C01836=1155.054,198.097,-61.668,-178.059,7.198,148.783
C01837=1155.049,198.346,-61.692,-178.056,7.200,148.783
C01838=1155.045,198.596,-61.716,-178.053,7.203,148.783
C01839=1155.041,198.844,-61.740,-178.051,7.205,148.782
C01840=1155.036,199.093,-61.764,-178.048,7.208,148.782
C01841=1155.031,199.342,-61.788,-178.045,7.210,148.782
C01842=1155.027,199.590,-61.812,-178.042,7.213,148.782
C01843=1155.022,199.839,-61.836,-178.040,7.214,148.781
C01844=1155.018,200.088,-61.860,-178.037,7.217,148.781
C01845=1155.013,200.337,-61.885,-178.034,7.219,148.781
C01846=1155.009,200.585,-61.909,-178.032,7.222,148.781
C01847=1155.004,200.834,-61.932,-178.029,7.224,148.780
C01848=1155.000,201.083,-61.956,-178.026,7.227,148.780
C01849=1154.995,201.332,-61.981,-178.023,7.228,148.780
C01850=1154.991,201.581,-62.005,-178.021,7.231,148.780
C01851=1154.986,201.829,-62.029,-178.018,7.233,148.780
C01852=1154.981,202.078,-62.053,-178.015,7.236,148.779
C01853=1154.977,202.328,-62.078,-178.012,7.238,148.779
C01854=1154.973,202.576,-62.102,-178.010,7.241,148.779
C01855=1154.968,202.825,-62.127,-178.007,7.242,148.779
C01856=1154.963,203.073,-62.151,-178.004,7.245,148.779
C01857=1154.959,203.321,-62.175,-178.001,7.248,148.778
C01858=1154.954,203.572,-62.199,-177.999,7.250,148.778
C01859=1154.950,203.820,-62.223,-177.995,7.253,148.778
C01860=1154.945,204.068,-62.247,-177.993,7.255,148.778
C01861=1154.941,204.318,-62.272,-177.990,7.257,148.777
C01862=1154.936,204.566,-62.296,-177.988,7.259,148.777
C01863=1154.931,204.815,-62.321,-177.985,7.262,148.777
C01864=1154.927,205.063,-62.345,-177.982,7.264,148.777
C01865=1154.923,205.312,-62.369,-177.979,7.267,148.776
C01866=1154.918,205.561,-62.394,-177.977,7.269,148.776
C01867=1154.913,205.810,-62.418,-177.974,7.271,148.776
C01868=1154.909,206.059,-62.443,-177.971,7.273,148.776
C01869=1154.904,206.307,-62.467,-177.968,7.276,148.776
C01870=1154.899,206.556,-62.492,-177.965,7.279,148.775
C01871=1154.895,206.805,-62.516,-177.963,7.281,148.775
C01872=1154.890,207.054,-62.541,-177.960,7.284,148.775
C01873=1154.886,207.302,-62.565,-177.957,7.285,148.775
C01874=1154.881,207.551,-62.590,-177.954,7.288,148.775
C01875=1154.877,207.800,-62.614,-177.952,7.290,148.774
C01876=1154.872,208.049,-62.639,-177.949,7.293,148.774
C01877=1154.868,208.297,-62.664,-177.946,7.295,148.774
C01878=1154.863,208.546,-62.689,-177.943,7.298,148.774
C01879=1154.859,208.795,-62.713,-177.941,7.301,148.774
C01880=1154.854,209.044,-62.738,-177.938,7.302,148.773
C01881=1154.849,209.293,-62.763,-177.935,7.305,148.773
C01882=1154.844,209.563,-62.789,-177.932,7.308,148.773
C01883=1154.840,209.834,-62.816,-177.930,7.310,148.773
C01884=1154.834,210.104,-62.843,-177.926,7.312,148.772
C01885=1154.830,210.375,-62.870,-177.923,7.315,148.772
C01886=1154.825,210.623,-62.894,-177.920,7.318,148.772
C01887=1154.821,210.873,-62.919,-177.918,7.320,148.772
C01888=1154.816,211.121,-62.945,-177.915,7.323,148.772
C01889=1154.812,211.369,-62.969,-177.912,7.326,148.771
C01890=1154.807,211.619,-62.994,-177.910,7.327,148.771
C01891=1154.803,211.866,-63.019,-177.907,7.330,148.771
C01892=1154.799,212.116,-63.044,-177.904,7.332,148.771
C01893=1154.793,212.365,-63.068,-177.901,7.335,148.771
C01894=1154.789,212.612,-63.093,-177.898,7.338,148.770
C01895=1154.785,212.862,-63.118,-177.896,7.340,148.770
C01896=1154.780,213.110,-63.143,-177.893,7.343,148.770
C01897=1154.775,213.359,-63.169,-177.890,7.344,148.770
C01898=1154.771,213.608,-63.193,-177.888,7.347,148.770
C01899=1154.767,213.857,-63.218,-177.885,7.350,148.769
C01900=1154.762,214.105,-63.243,-177.882,7.352,148.769
C01901=1154.758,214.354,-63.267,-177.879,7.355,148.769
C01902=1154.753,214.602,-63.293,-177.877,7.357,148.769
C01903=1154.749,214.852,-63.318,-177.874,7.360,148.769
C01904=1154.744,215.100,-63.343,-177.871,7.363,148.769
C01905=1154.740,215.349,-63.368,-177.868,7.364,148.768
C01906=1154.735,215.597,-63.393,-177.866,7.367,148.768
C01907=1154.731,215.847,-63.418,-177.863,7.369,148.768
C01908=1154.726,216.095,-63.443,-177.860,7.372,148.768
C01909=1154.722,216.344,-63.468,-177.857,7.375,148.768
C01910=1154.717,216.592,-63.493,-177.855,7.377,148.767
C01911=1154.713,216.841,-63.518,-177.852,7.380,148.767
C01912=1154.708,217.089,-63.544,-177.849,7.382,148.767
C01913=1154.703,217.339,-63.569,-177.846,7.384,148.767
C01914=1154.698,217.587,-63.594,-177.844,7.387,148.767
C01915=1154.695,217.835,-63.619,-177.840,7.390,148.766
C01916=1154.690,218.085,-63.644,-177.838,7.392,148.766
C01917=1154.686,218.333,-63.670,-177.835,7.395,148.766
C01918=1154.681,218.582,-63.695,-177.833,7.397,148.766
C01919=1154.676,218.831,-63.720,-177.830,7.399,148.766
C01920=1154.672,219.079,-63.746,-177.827,7.402,148.766
C01921=1154.667,219.327,-63.771,-177.824,7.404,148.765
C01922=1154.663,219.577,-63.796,-177.822,7.407,148.765
C01923=1154.659,219.825,-63.821,-177.819,7.410,148.765
C01924=1154.654,220.073,-63.847,-177.816,7.412,148.765
C01925=1154.650,220.323,-63.872,-177.813,7.415,148.765
C01926=1154.645,220.571,-63.897,-177.811,7.418,148.765
C01927=1154.641,220.820,-63.923,-177.808,7.419,148.764
C01928=1154.637,221.069,-63.949,-177.805,7.422,148.764
C01929=1154.631,221.317,-63.973,-177.802,7.425,148.764
C01930=1154.627,221.566,-63.999,-177.800,7.427,148.764
C01931=1154.623,221.815,-64.025,-177.797,7.430,148.764
C01932=1154.618,222.063,-64.050,-177.794,7.433,148.763
C01933=1154.614,222.312,-64.076,-177.792,7.435,148.763
C01934=1154.609,222.560,-64.101,-177.789,7.438,148.763
C01935=1154.605,222.809,-64.127,-177.786,7.441,148.763
C01936=1154.600,223.058,-64.152,-177.783,7.442,148.763
C01937=1154.595,223.306,-64.178,-177.780,7.445,148.763
C01938=1154.591,223.555,-64.203,-177.778,7.448,148.762
C01939=1154.587,223.804,-64.229,-177.775,7.450,148.762
C01940=1154.582,224.052,-64.255,-177.772,7.453,148.762
C01941=1154.578,224.301,-64.280,-177.769,7.456,148.762
C01942=1154.574,224.550,-64.306,-177.766,7.458,148.762
C01943=1154.570,224.798,-64.332,-177.764,7.460,148.762
C01944=1154.565,225.047,-64.357,-177.761,7.463,148.761
C01945=1154.560,225.296,-64.384,-177.758,7.466,148.761
C01946=1154.556,225.544,-64.409,-177.756,7.468,148.761
C01947=1154.551,225.793,-64.435,-177.753,7.471,148.761
C01948=1154.546,226.041,-64.460,-177.750,7.474,148.761
C01949=1154.542,226.290,-64.486,-177.748,7.476,148.761
C01950=1154.538,226.539,-64.512,-177.745,7.479,148.760
C01951=1154.533,226.787,-64.537,-177.742,7.482,148.760
C01952=1154.529,227.036,-64.563,-177.739,7.484,148.760
C01953=1154.524,227.285,-64.589,-177.737,7.486,148.760
C01954=1154.520,227.534,-64.615,-177.734,7.489,148.760
C01955=1154.515,227.782,-64.641,-177.731,7.492,148.760
C01956=1154.511,228.031,-64.666,-177.728,7.494,148.759
C01957=1154.507,228.279,-64.693,-177.725,7.497,148.759
C01958=1154.502,228.528,-64.719,-177.723,7.500,148.759
C01959=1154.497,228.776,-64.744,-177.720,7.503,148.759
C01960=1154.493,229.025,-64.770,-177.717,7.505,148.759
C01961=1154.489,229.274,-64.796,-177.714,7.507,148.759
C01962=1154.484,229.523,-64.822,-177.712,7.510,148.759
C01963=1154.480,229.771,-64.849,-177.709,7.513,148.759
C01964=1154.475,230.019,-64.874,-177.706,7.515,148.758
C01965=1154.471,230.268,-64.900,-177.703,7.518,148.758
C01966=1154.466,230.517,-64.926,-177.701,7.521,148.758
C01967=1154.462,230.765,-64.953,-177.698,7.523,148.758
C01968=1154.458,231.014,-64.978,-177.695,7.526,148.758
C01969=1154.453,231.263,-65.004,-177.692,7.529,148.758
C01970=1154.448,231.511,-65.031,-177.690,7.532,148.758
C01971=1154.444,231.759,-65.057,-177.687,7.534,148.757
C01972=1154.440,232.008,-65.082,-177.684,7.536,148.757
C01973=1154.435,232.257,-65.109,-177.681,7.539,148.757
C01974=1154.431,232.506,-65.135,-177.679,7.542,148.757
C01975=1154.427,232.754,-65.161,-177.676,7.544,148.757
C01976=1154.422,233.003,-65.188,-177.673,7.547,148.757
C01977=1154.417,233.251,-65.213,-177.670,7.550,148.756
C01978=1154.413,233.499,-65.240,-177.668,7.553,148.756
C01979=1154.408,233.748,-65.266,-177.665,7.556,148.756
C01980=1154.404,233.997,-65.292,-177.663,7.558,148.756
C01981=1154.399,234.246,-65.319,-177.659,7.560,148.756
C01982=1154.395,234.494,-65.345,-177.657,7.563,148.756
C01983=1154.391,234.743,-65.371,-177.654,7.566,148.756
C01984=1154.386,234.992,-65.398,-177.652,7.568,148.756
C01985=1154.382,235.240,-65.424,-177.648,7.571,148.755
C01986=1154.377,235.512,-65.453,-177.646,7.574,148.755
C01987=1154.372,235.783,-65.481,-177.643,7.577,148.755
C01988=1154.367,236.055,-65.511,-177.640,7.580,148.755
C01989=1154.362,236.327,-65.539,-177.636,7.583,148.755
C01990=1154.358,236.575,-65.566,-177.634,7.585,148.755
C01991=1154.353,236.824,-65.592,-177.631,7.588,148.755
C01992=1154.349,237.073,-65.619,-177.628,7.591,148.755
C01993=1154.344,237.321,-65.646,-177.626,7.594,148.754
C01994=1154.340,237.570,-65.672,-177.622,7.597,148.754
C01995=1154.336,237.818,-65.699,-177.620,7.599,148.754
C01996=1154.332,238.067,-65.725,-177.617,7.602,148.754
C01997=1154.327,238.316,-65.751,-177.615,7.605,148.754
C01998=1154.323,238.564,-65.778,-177.612,7.608,148.754
C01999=1154.318,238.812,-65.805,-177.609,7.610,148.754
C02000=1154.314,239.061,-65.831,-177.606,7.612,148.753
C02001=1154.309,239.310,-65.858,-177.604,7.615,148.753
C02002=1154.305,239.558,-65.884,-177.601,7.618,148.753
C02003=1154.300,239.807,-65.911,-177.598,7.621,148.753
C02004=1154.296,240.056,-65.938,-177.595,7.624,148.753
C02005=1154.292,240.304,-65.964,-177.593,7.626,148.753
C02006=1154.287,240.552,-65.991,-177.590,7.629,148.753
C02007=1154.282,240.801,-66.018,-177.587,7.632,148.753
C02008=1154.278,241.049,-66.044,-177.584,7.635,148.753
C02009=1154.274,241.298,-66.071,-177.582,7.637,148.753
C02010=1154.270,241.546,-66.098,-177.579,7.640,148.752
C02011=1154.265,241.795,-66.125,-177.577,7.643,148.752
C02012=1154.260,242.043,-66.152,-177.574,7.645,148.752
C02013=1154.256,242.291,-66.178,-177.571,7.648,148.752
C02014=1154.252,242.540,-66.205,-177.568,7.651,148.752
C02015=1154.247,242.789,-66.232,-177.565,7.654,148.752
C02016=1154.242,243.037,-66.259,-177.563,7.656,148.752
C02017=1154.238,243.286,-66.285,-177.560,7.659,148.752
C02018=1154.234,243.535,-66.312,-177.557,7.662,148.752
C02019=1154.229,243.783,-66.340,-177.555,7.665,148.751
C02020=1154.226,244.032,-66.366,-177.552,7.668,148.751
C02021=1154.221,244.280,-66.393,-177.548,7.670,148.751
C02022=1154.216,244.528,-66.420,-177.546,7.673,148.751
C02023=1154.212,244.777,-66.447,-177.544,7.675,148.751
C02024=1154.207,245.025,-66.474,-177.541,7.678,148.751
C02025=1154.203,245.274,-66.501,-177.538,7.681,148.751
C02026=1154.199,245.523,-66.528,-177.535,7.684,148.751
C02027=1154.194,245.771,-66.555,-177.532,7.687,148.751
C02028=1154.190,246.020,-66.582,-177.530,7.689,148.751
C02029=1154.186,246.268,-66.609,-177.527,7.692,148.750
C02030=1154.181,246.516,-66.637,-177.525,7.695,148.750
C02031=1154.177,246.764,-66.664,-177.521,7.698,148.750
C02032=1154.172,247.013,-66.691,-177.519,7.701,148.750
C02033=1154.168,247.262,-66.718,-177.516,7.704,148.750
C02034=1154.163,247.511,-66.745,-177.513,7.707,148.750
C02035=1154.159,247.759,-66.772,-177.511,7.709,148.750
C02036=1154.155,248.007,-66.799,-177.508,7.712,148.750
C02037=1154.150,248.255,-66.826,-177.505,7.715,148.750
C02038=1154.146,248.504,-66.854,-177.503,7.718,148.750
C02039=1154.142,248.753,-66.881,-177.500,7.720,148.750
C02040=1154.137,249.001,-66.908,-177.497,7.723,148.749
C02041=1154.133,249.249,-66.936,-177.494,7.726,148.749
C02042=1154.128,249.498,-66.963,-177.491,7.729,148.749
C02043=1154.124,249.747,-66.990,-177.489,7.731,148.749
C02044=1154.119,249.995,-67.017,-177.486,7.734,148.749
C02045=1154.115,250.243,-67.045,-177.483,7.737,148.749
C02046=1154.110,250.492,-67.072,-177.480,7.740,148.749
C02047=1154.106,250.741,-67.100,-177.478,7.743,148.749
C02048=1154.102,250.989,-67.127,-177.475,7.746,148.749
C02049=1154.097,251.237,-67.154,-177.472,7.749,148.749
C02050=1154.093,251.486,-67.181,-177.469,7.752,148.749
C02051=1154.089,251.734,-67.210,-177.467,7.754,148.748
C02052=1154.084,251.983,-67.237,-177.464,7.757,148.748
C02053=1154.080,252.231,-67.264,-177.462,7.760,148.748
C02054=1154.076,252.480,-67.292,-177.459,7.763,148.748
C02055=1154.071,252.728,-67.319,-177.456,7.765,148.748
C02056=1154.067,252.976,-67.347,-177.453,7.768,148.748
C02057=1154.062,253.225,-67.374,-177.451,7.771,148.748
C02058=1154.058,253.473,-67.402,-177.448,7.774,148.748
C02059=1154.054,253.722,-67.429,-177.445,7.777,148.748
C02060=1154.049,253.970,-67.457,-177.442,7.780,148.748
C02061=1154.045,254.219,-67.484,-177.440,7.782,148.748
C02062=1154.041,254.467,-67.512,-177.437,7.785,148.748
C02063=1154.036,254.715,-67.539,-177.434,7.788,148.748
C02064=1154.032,254.964,-67.568,-177.432,7.791,148.748
C02065=1154.027,255.213,-67.595,-177.429,7.794,148.747
C02066=1154.023,255.461,-67.623,-177.426,7.797,148.747
C02067=1154.019,255.709,-67.651,-177.423,7.800,148.747
C02068=1154.014,255.958,-67.678,-177.421,7.803,148.747
C02069=1154.011,256.206,-67.706,-177.418,7.806,148.747
C02070=1154.006,256.455,-67.733,-177.415,7.809,148.747
C02071=1154.001,256.703,-67.761,-177.412,7.812,148.747
C02072=1153.997,256.952,-67.790,-177.410,7.814,148.747
C02073=1153.993,257.200,-67.817,-177.407,7.817,148.747
C02074=1153.988,257.448,-67.844,-177.404,7.820,148.747
C02075=1153.984,257.696,-67.873,-177.402,7.823,148.747
C02076=1153.979,257.945,-67.901,-177.399,7.826,148.747
C02077=1153.975,258.194,-67.928,-177.396,7.829,148.747
C02078=1153.971,258.442,-67.956,-177.393,7.831,148.747
C02079=1153.967,258.690,-67.984,-177.391,7.834,148.747
C02080=1153.962,258.939,-68.012,-177.388,7.837,148.747
C02081=1153.957,259.187,-68.040,-177.385,7.840,148.746
C02082=1153.954,259.436,-68.068,-177.383,7.844,148.747
C02083=1153.949,259.683,-68.096,-177.380,7.846,148.747
C02084=1153.945,259.932,-68.124,-177.377,7.849,148.746
C02085=1153.940,260.180,-68.152,-177.374,7.852,148.746
C02086=1153.936,260.429,-68.180,-177.372,7.855,148.746
C02087=1153.931,260.678,-68.208,-177.369,7.858,148.746
C02088=1153.928,260.926,-68.236,-177.367,7.860,148.746
C02089=1153.923,261.174,-68.264,-177.364,7.863,148.746
C02090=1153.918,261.448,-68.295,-177.361,7.867,148.746
C02091=1153.913,261.721,-68.326,-177.358,7.870,148.746
C02092=1153.909,261.994,-68.356,-177.355,7.873,148.746
C02093=1153.904,262.267,-68.388,-177.352,7.877,148.746
C02094=1153.900,262.516,-68.417,-177.349,7.880,148.746
C02095=1153.895,262.764,-68.444,-177.346,7.883,148.746
C02096=1153.892,263.012,-68.472,-177.343,7.886,148.746
C02097=1153.886,263.261,-68.501,-177.341,7.888,148.746
C02098=1153.883,263.509,-68.529,-177.338,7.891,148.746
C02099=1153.878,263.757,-68.557,-177.335,7.894,148.746
C02100=1153.874,264.006,-68.586,-177.333,7.898,148.746
C02101=1153.869,264.254,-68.614,-177.331,7.900,148.746
C02102=1153.865,264.503,-68.642,-177.328,7.903,148.746
C02103=1153.860,264.751,-68.670,-177.325,7.906,148.746
C02104=1153.856,264.999,-68.699,-177.322,7.909,148.746
C02105=1153.852,265.247,-68.726,-177.319,7.912,148.745
C02106=1153.847,265.496,-68.755,-177.317,7.914,148.745
C02107=1153.844,265.745,-68.783,-177.314,7.917,148.745
C02108=1153.839,265.993,-68.812,-177.311,7.920,148.745
C02109=1153.834,266.241,-68.841,-177.309,7.924,148.745
C02110=1153.830,266.489,-68.869,-177.306,7.927,148.745
C02111=1153.826,266.738,-68.898,-177.303,7.930,148.745
C02112=1153.821,266.986,-68.925,-177.300,7.932,148.745
C02113=1153.817,267.235,-68.954,-177.298,7.935,148.745
C02114=1153.813,267.483,-68.983,-177.295,7.938,148.745
C02115=1153.808,267.731,-69.011,-177.292,7.941,148.745
C02116=1153.804,267.980,-69.039,-177.290,7.945,148.745
C02117=1153.799,268.228,-69.068,-177.287,7.948,148.745
C02118=1153.795,268.476,-69.097,-177.284,7.950,148.745
C02119=1153.791,268.725,-69.125,-177.282,7.953,148.745
C02120=1153.786,268.973,-69.154,-177.279,7.956,148.745
C02121=1153.783,269.221,-69.182,-177.276,7.959,148.745
C02122=1153.778,269.470,-69.211,-177.273,7.962,148.745
C02123=1153.773,269.718,-69.240,-177.271,7.966,148.745
C02124=1153.770,269.966,-69.269,-177.268,7.968,148.745
C02125=1153.765,270.215,-69.297,-177.265,7.971,148.745
C02126=1153.760,270.463,-69.326,-177.263,7.974,148.745
C02127=1153.757,270.711,-69.355,-177.260,7.977,148.745
C02128=1153.752,270.960,-69.383,-177.258,7.981,148.745
C02129=1153.748,271.207,-69.412,-177.255,7.983,148.745
C02130=1153.744,271.456,-69.441,-177.252,7.986,148.745
C02131=1153.739,271.705,-69.469,-177.249,7.989,148.745
C02132=1153.735,271.952,-69.498,-177.246,7.992,148.745
C02133=1153.730,272.201,-69.527,-177.244,7.995,148.745
C02134=1153.727,272.449,-69.556,-177.241,7.999,148.745
C02135=1153.722,272.698,-69.585,-177.239,8.001,148.745
C02136=1153.717,272.946,-69.614,-177.236,8.004,148.745
C02137=1153.713,273.194,-69.643,-177.233,8.007,148.745
C02138=1153.709,273.442,-69.671,-177.231,8.011,148.745
C02139=1153.705,273.691,-69.701,-177.228,8.014,148.745
C02140=1153.700,273.939,-69.729,-177.225,8.017,148.745
C02141=1153.696,274.187,-69.759,-177.222,8.019,148.745
C02142=1153.692,274.436,-69.787,-177.220,8.022,148.745
C02143=1153.688,274.684,-69.816,-177.217,8.026,148.745
C02144=1153.683,274.931,-69.845,-177.214,8.029,148.745
C02145=1153.679,275.180,-69.874,-177.211,8.032,148.745
C02146=1153.675,275.429,-69.904,-177.208,8.035,148.745
C02147=1153.670,275.677,-69.933,-177.206,8.039,148.745
C02148=1153.667,275.926,-69.961,-177.203,8.042,148.745
C02149=1153.662,276.173,-69.990,-177.201,8.045,148.745
C02150=1153.658,276.421,-70.020,-177.198,8.047,148.745
C02151=1153.653,276.670,-70.049,-177.196,8.051,148.745
C02152=1153.649,276.918,-70.078,-177.193,8.054,148.745
C02153=1153.645,277.167,-70.107,-177.190,8.057,148.745
C02154=1153.640,277.414,-70.136,-177.187,8.060,148.745
C02155=1153.636,277.663,-70.166,-177.185,8.063,148.745
C02156=1153.632,277.911,-70.194,-177.182,8.066,148.745
C02157=1153.628,278.159,-70.223,-177.179,8.069,148.745
C02158=1153.624,278.408,-70.253,-177.177,8.072,148.745
C02159=1153.620,278.656,-70.282,-177.174,8.075,148.745
C02160=1153.615,278.904,-70.312,-177.171,8.078,148.745
C02161=1153.611,279.152,-70.341,-177.169,8.081,148.745
C02162=1153.606,279.401,-70.370,-177.166,8.084,148.745
C02163=1153.602,279.649,-70.399,-177.164,8.087,148.745
C02164=1153.598,279.897,-70.429,-177.161,8.090,148.745
C02165=1153.594,280.145,-70.458,-177.158,8.094,148.745
C02166=1153.589,280.394,-70.487,-177.155,8.097,148.745
C02167=1153.585,280.642,-70.517,-177.152,8.100,148.745
C02168=1153.581,280.890,-70.546,-177.150,8.103,148.745
C02169=1153.577,281.139,-70.576,-177.147,8.106,148.745
C02170=1153.572,281.386,-70.605,-177.145,8.109,148.745
C02171=1153.568,281.634,-70.634,-177.142,8.112,148.745
C02172=1153.564,281.883,-70.664,-177.140,8.115,148.745
C02173=1153.559,282.131,-70.694,-177.137,8.118,148.745
C02174=1153.555,282.380,-70.723,-177.134,8.121,148.745
C02175=1153.550,282.628,-70.753,-177.131,8.124,148.745
C02176=1153.546,282.876,-70.782,-177.129,8.128,148.745
C02177=1153.542,283.124,-70.812,-177.126,8.130,148.745
C02178=1153.538,283.373,-70.841,-177.123,8.133,148.745
C02179=1153.534,283.620,-70.871,-177.120,8.137,148.745
C02180=1153.530,283.868,-70.901,-177.118,8.140,148.745
C02181=1153.526,284.117,-70.930,-177.115,8.143,148.745
C02182=1153.521,284.365,-70.960,-177.113,8.147,148.746
C02183=1153.517,284.614,-70.990,-177.110,8.150,148.745
C02184=1153.512,284.862,-71.019,-177.108,8.153,148.746
C02185=1153.508,285.110,-71.049,-177.105,8.156,148.746
C02186=1153.504,285.358,-71.079,-177.102,8.159,148.746
C02187=1153.499,285.606,-71.109,-177.100,8.162,148.746
C02188=1153.495,285.855,-71.138,-177.097,8.165,148.746
C02189=1153.491,286.103,-71.168,-177.094,8.169,148.746
C02190=1153.487,286.351,-71.198,-177.091,8.172,148.746
C02191=1153.483,286.599,-71.227,-177.088,8.175,148.746
C02192=1153.478,286.847,-71.257,-177.086,8.178,148.746
C02193=1153.474,287.095,-71.288,-177.083,8.181,148.746
C02194=1153.469,287.370,-71.320,-177.081,8.184,148.746
C02195=1153.465,287.645,-71.353,-177.077,8.188,148.746
C02196=1153.460,287.921,-71.386,-177.074,8.192,148.746
C02197=1153.456,288.196,-71.420,-177.072,8.195,148.746
C02198=1153.451,288.445,-71.450,-177.069,8.198,148.746
C02199=1153.447,288.692,-71.480,-177.067,8.201,148.746
C02200=1153.443,288.941,-71.509,-177.064,8.204,148.746
C02201=1153.438,289.189,-71.539,-177.061,8.208,148.746
C02202=1153.434,289.437,-71.570,-177.058,8.211,148.746
C02203=1153.430,289.685,-71.599,-177.056,8.214,148.747
C02204=1153.425,289.933,-71.630,-177.053,8.217,148.746
C02205=1153.421,290.181,-71.659,-177.050,8.220,148.746
C02206=1153.417,290.429,-71.690,-177.048,8.224,148.747
C02207=1153.412,290.677,-71.720,-177.045,8.227,148.747
C02208=1153.409,290.926,-71.750,-177.043,8.230,148.747
C02209=1153.405,291.174,-71.780,-177.040,8.234,148.747
C02210=1153.400,291.422,-71.810,-177.037,8.237,148.747
C02211=1153.396,291.670,-71.840,-177.034,8.240,148.747
C02212=1153.391,291.918,-71.871,-177.032,8.243,148.747
C02213=1153.387,292.167,-71.900,-177.029,8.246,148.747
C02214=1153.382,292.415,-71.931,-177.027,8.249,148.747
C02215=1153.379,292.663,-71.961,-177.024,8.252,148.747
C02216=1153.375,292.911,-71.991,-177.021,8.256,148.747
C02217=1153.370,293.159,-72.021,-177.019,8.259,148.747
C02218=1153.366,293.407,-72.052,-177.016,8.262,148.747
C02219=1153.362,293.655,-72.082,-177.014,8.266,148.747
C02220=1153.358,293.903,-72.112,-177.011,8.269,148.747
C02221=1153.354,294.152,-72.143,-177.008,8.272,148.748
C02222=1153.349,294.400,-72.172,-177.006,8.275,148.748
C02223=1153.345,294.648,-72.203,-177.003,8.279,148.748
C02224=1153.341,294.895,-72.233,-177.000,8.282,148.748
C02225=1153.336,295.143,-72.264,-176.998,8.285,148.748
C02226=1153.333,295.392,-72.294,-176.995,8.288,148.748
C02227=1153.328,295.640,-72.325,-176.992,8.291,148.748
C02228=1153.324,295.888,-72.355,-176.990,8.294,148.748
C02229=1153.320,296.136,-72.386,-176.987,8.297,148.748
C02230=1153.316,296.385,-72.417,-176.984,8.301,148.748
C02231=1153.311,296.633,-72.446,-176.981,8.304,148.748
C02232=1153.307,296.881,-72.477,-176.979,8.308,148.748
C02233=1153.303,297.128,-72.507,-176.977,8.311,148.749
C02234=1153.299,297.377,-72.538,-176.974,8.314,148.749
C02235=1153.294,297.625,-72.569,-176.972,8.317,148.749
C02236=1153.290,297.873,-72.599,-176.968,8.321,148.749
C02237=1153.286,298.121,-72.630,-176.966,8.324,148.749
C02238=1153.282,298.369,-72.661,-176.963,8.327,148.749
C02239=1153.278,298.617,-72.691,-176.961,8.330,148.749
C02240=1153.273,298.865,-72.722,-176.958,8.333,148.749
C02241=1153.269,299.114,-72.753,-176.955,8.337,148.749
C02242=1153.265,299.361,-72.783,-176.953,8.340,148.749
C02243=1153.261,299.609,-72.814,-176.950,8.344,148.749
C02244=1153.256,299.857,-72.845,-176.948,8.347,148.749
C02245=1153.253,300.106,-72.875,-176.945,8.350,148.749
C02246=1153.248,300.354,-72.906,-176.942,8.353,148.749
C02247=1153.244,300.601,-72.937,-176.940,8.357,148.750
C02248=1153.240,300.850,-72.968,-176.937,8.360,148.750
C02249=1153.236,301.098,-72.998,-176.934,8.363,148.750
C02250=1153.231,301.346,-73.029,-176.932,8.366,148.750
C02251=1153.227,301.594,-73.060,-176.929,8.369,148.750
C02252=1153.223,301.842,-73.091,-176.926,8.373,148.750
C02253=1153.219,302.090,-73.121,-176.924,8.376,148.750
C02254=1153.215,302.338,-73.153,-176.921,8.380,148.750
C02255=1153.210,302.586,-73.184,-176.919,8.383,148.751
C02256=1153.206,302.835,-73.215,-176.916,8.386,148.750
C02257=1153.202,303.083,-73.246,-176.913,8.390,148.751
C02258=1153.197,303.331,-73.276,-176.911,8.393,148.751
C02259=1153.194,303.579,-73.307,-176.908,8.396,148.751
C02260=1153.190,303.826,-73.338,-176.906,8.399,148.751
C02261=1153.185,304.074,-73.369,-176.903,8.402,148.751
C02262=1153.181,304.323,-73.400,-176.900,8.406,148.751
C02263=1153.177,304.570,-73.432,-176.898,8.409,148.751
C02264=1153.173,304.819,-73.463,-176.895,8.413,148.751
C02265=1153.168,305.067,-73.494,-176.893,8.416,148.752
C02266=1153.163,305.315,-73.524,-176.890,8.419,148.752
C02267=1153.160,305.563,-73.556,-176.887,8.423,148.752
C02268=1153.156,305.810,-73.586,-176.885,8.426,148.752
C02269=1153.152,306.059,-73.618,-176.882,8.429,148.752
C02270=1153.148,306.306,-73.649,-176.880,8.433,148.752
C02271=1153.144,306.555,-73.680,-176.877,8.436,148.752
C02272=1153.139,306.802,-73.712,-176.874,8.440,148.752
C02273=1153.135,307.051,-73.743,-176.872,8.443,148.752
C02274=1153.131,307.299,-73.774,-176.869,8.446,148.752
C02275=1153.126,307.546,-73.805,-176.867,8.449,148.753
C02276=1153.122,307.795,-73.836,-176.864,8.453,148.753
C02277=1153.118,308.042,-73.868,-176.861,8.456,148.753
C02278=1153.114,308.291,-73.899,-176.859,8.459,148.753
C02279=1153.110,308.538,-73.930,-176.857,8.463,148.753
C02280=1153.106,308.787,-73.961,-176.853,8.466,148.753
C02281=1153.101,309.034,-73.993,-176.851,8.470,148.753
C02282=1153.097,309.283,-74.024,-176.849,8.473,148.754
C02283=1153.093,309.530,-74.055,-176.846,8.476,148.754
C02284=1153.089,309.778,-74.087,-176.843,8.480,148.754
C02285=1153.085,310.027,-74.118,-176.841,8.483,148.754
C02286=1153.080,310.275,-74.150,-176.838,8.486,148.754
C02287=1153.076,310.523,-74.182,-176.836,8.490,148.754
C02288=1153.072,310.771,-74.213,-176.833,8.494,148.754
C02289=1153.068,311.019,-74.245,-176.830,8.497,148.755
C02290=1153.064,311.267,-74.276,-176.828,8.500,148.755
C02291=1153.060,311.515,-74.308,-176.825,8.503,148.755
C02292=1153.056,311.762,-74.339,-176.822,8.507,148.755
C02293=1153.052,312.011,-74.370,-176.820,8.510,148.755
C02294=1153.048,312.259,-74.402,-176.817,8.513,148.755
C02295=1153.043,312.506,-74.434,-176.815,8.517,148.755
C02296=1153.039,312.755,-74.466,-176.812,8.521,148.756
C02297=1153.034,313.002,-74.497,-176.809,8.524,148.755
C02298=1153.030,313.280,-74.532,-176.806,8.528,148.756
C02299=1153.026,313.558,-74.568,-176.804,8.531,148.756
C02300=1153.021,313.834,-74.603,-176.801,8.535,148.756
C02301=1153.017,314.112,-74.639,-176.798,8.539,148.756
C02302=1153.012,314.361,-74.670,-176.796,8.542,148.756
C02303=1153.008,314.608,-74.702,-176.793,8.546,148.757
C02304=1153.004,314.856,-74.734,-176.790,8.549,148.757
C02305=1153.000,315.104,-74.766,-176.788,8.553,148.757
C02306=1152.995,315.352,-74.798,-176.785,8.556,148.757
C02307=1152.991,315.600,-74.830,-176.782,8.560,148.757
C02308=1152.988,315.848,-74.861,-176.780,8.563,148.757
C02309=1152.983,316.095,-74.893,-176.777,8.566,148.757
C02310=1152.979,316.344,-74.925,-176.775,8.569,148.758
C02311=1152.975,316.592,-74.957,-176.772,8.574,148.758
C02312=1152.971,316.839,-74.989,-176.770,8.577,148.758
C02313=1152.966,317.087,-75.021,-176.767,8.580,148.758
C02314=1152.963,317.335,-75.053,-176.764,8.584,148.758
C02315=1152.958,317.583,-75.084,-176.762,8.587,148.758
C02316=1152.954,317.831,-75.117,-176.759,8.590,148.759
C02317=1152.950,318.079,-75.149,-176.757,8.593,148.759
C02318=1152.947,318.327,-75.181,-176.754,8.598,148.759
C02319=1152.942,318.575,-75.213,-176.752,8.601,148.759
C02320=1152.938,318.823,-75.244,-176.749,8.604,148.759
C02321=1152.934,319.071,-75.276,-176.746,8.608,148.759
C02322=1152.929,319.319,-75.308,-176.744,8.611,148.760
C02323=1152.925,319.567,-75.340,-176.741,8.614,148.760
C02324=1152.921,319.815,-75.373,-176.738,8.618,148.760
C02325=1152.918,320.062,-75.405,-176.736,8.622,148.760
C02326=1152.913,320.310,-75.437,-176.734,8.625,148.760
C02327=1152.909,320.558,-75.469,-176.731,8.628,148.760
C02328=1152.905,320.806,-75.501,-176.728,8.632,148.760
C02329=1152.901,321.054,-75.533,-176.726,8.635,148.761
C02330=1152.897,321.302,-75.566,-176.723,8.639,148.761
C02331=1152.892,321.550,-75.598,-176.721,8.643,148.761
C02332=1152.889,321.798,-75.630,-176.718,8.646,148.761
C02333=1152.884,322.046,-75.662,-176.716,8.649,148.761
C02334=1152.881,322.293,-75.695,-176.713,8.653,148.762
C02335=1152.876,322.542,-75.727,-176.710,8.656,148.762
C02336=1152.872,322.789,-75.759,-176.708,8.660,148.762
C02337=1152.868,323.037,-75.792,-176.705,8.664,148.762
C02338=1152.864,323.285,-75.824,-176.703,8.667,148.762
C02339=1152.860,323.533,-75.856,-176.700,8.670,148.762
C02340=1152.856,323.781,-75.889,-176.697,8.674,148.763
C02341=1152.852,324.029,-75.921,-176.695,8.678,148.763
C02342=1152.848,324.276,-75.953,-176.693,8.681,148.763
C02343=1152.843,324.524,-75.986,-176.690,8.685,148.763
C02344=1152.839,324.772,-76.018,-176.687,8.688,148.763
C02345=1152.835,325.020,-76.051,-176.685,8.691,148.763
C02346=1152.831,325.268,-76.083,-176.682,8.695,148.764
C02347=1152.828,325.516,-76.116,-176.680,8.699,148.764
C02348=1152.823,325.764,-76.148,-176.677,8.702,148.764
C02349=1152.818,326.011,-76.181,-176.674,8.706,148.764
C02350=1152.815,326.259,-76.213,-176.672,8.709,148.764
C02351=1152.811,326.507,-76.246,-176.670,8.713,148.765
C02352=1152.806,326.755,-76.279,-176.667,8.717,148.765
C02353=1152.803,327.002,-76.311,-176.665,8.720,148.765
C02354=1152.798,327.251,-76.344,-176.662,8.723,148.765
C02355=1152.794,327.499,-76.377,-176.659,8.727,148.765
C02356=1152.791,327.746,-76.409,-176.657,8.730,148.766
C02357=1152.786,327.994,-76.442,-176.654,8.734,148.766
C02358=1152.782,328.242,-76.475,-176.651,8.738,148.766
C02359=1152.778,328.490,-76.508,-176.649,8.741,148.766
C02360=1152.774,328.737,-76.540,-176.646,8.745,148.766
C02361=1152.770,328.985,-76.573,-176.644,8.748,148.767
C02362=1152.765,329.233,-76.606,-176.642,8.751,148.767
C02363=1152.761,329.481,-76.638,-176.639,8.756,148.767
C02364=1152.758,329.728,-76.671,-176.636,8.759,148.767
C02365=1152.754,329.976,-76.704,-176.634,8.762,148.767
C02366=1152.749,330.224,-76.736,-176.631,8.766,148.768
C02367=1152.745,330.472,-76.770,-176.629,8.770,148.768
C02368=1152.741,330.720,-76.803,-176.626,8.774,148.768
C02369=1152.737,330.967,-76.835,-176.624,8.777,148.768
C02370=1152.733,331.215,-76.868,-176.621,8.780,148.769
C02371=1152.729,331.463,-76.901,-176.618,8.784,148.769
C02372=1152.725,331.711,-76.934,-176.616,8.788,148.769
C02373=1152.721,331.959,-76.967,-176.614,8.791,148.769
C02374=1152.716,332.207,-77.000,-176.611,8.795,148.769
C02375=1152.712,332.454,-77.034,-176.609,8.798,148.770
C02376=1152.709,332.702,-77.066,-176.606,8.802,148.770
C02377=1152.705,332.949,-77.099,-176.603,8.806,148.770
C02378=1152.700,333.198,-77.132,-176.601,8.809,148.770
C02379=1152.696,333.445,-77.165,-176.598,8.813,148.770
C02380=1152.692,333.693,-77.198,-176.596,8.816,148.771
C02381=1152.688,333.941,-77.231,-176.593,8.820,148.771
C02382=1152.684,334.189,-77.264,-176.591,8.824,148.771
C02383=1152.680,334.437,-77.298,-176.588,8.827,148.771
C02384=1152.676,334.685,-77.331,-176.585,8.831,148.772
C02385=1152.672,334.933,-77.364,-176.583,8.834,148.772
C02386=1152.668,335.180,-77.397,-176.580,8.838,148.772
C02387=1152.664,335.428,-77.430,-176.578,8.842,148.772
C02388=1152.659,335.676,-77.464,-176.575,8.845,148.772
C02389=1152.655,335.923,-77.497,-176.573,8.849,148.773
C02390=1152.652,336.171,-77.531,-176.570,8.852,148.773
C02391=1152.647,336.418,-77.564,-176.567,8.856,148.773
C02392=1152.643,336.666,-77.597,-176.565,8.860,148.774
C02393=1152.639,336.914,-77.630,-176.563,8.864,148.774
C02394=1152.636,337.162,-77.664,-176.560,8.867,148.774
C02395=1152.631,337.410,-77.697,-176.558,8.871,148.774
C02396=1152.627,337.658,-77.730,-176.555,8.875,148.774
C02397=1152.623,337.905,-77.764,-176.553,8.878,148.775
C02398=1152.619,338.152,-77.797,-176.550,8.882,148.775
C02399=1152.615,338.400,-77.830,-176.548,8.885,148.775
C02400=1152.611,338.648,-77.863,-176.545,8.889,148.775
C02401=1152.608,338.896,-77.897,-176.542,8.893,148.775
C02402=1152.602,339.176,-77.935,-176.539,8.897,148.776
C02403=1152.598,339.457,-77.973,-176.537,8.901,148.776
C02404=1152.594,339.736,-78.010,-176.534,8.905,148.776
C02405=1152.589,340.017,-78.049,-176.531,8.909,148.777
C02406=1152.585,340.264,-78.083,-176.529,8.913,148.777
C02407=1152.581,340.512,-78.116,-176.526,8.917,148.777
C02408=1152.577,340.759,-78.149,-176.524,8.920,148.777
C02409=1152.573,341.006,-78.183,-176.521,8.924,148.778
C02410=1152.569,341.255,-78.217,-176.518,8.927,148.778
C02411=1152.564,341.503,-78.250,-176.516,8.932,148.778
C02412=1152.561,341.750,-78.284,-176.514,8.935,148.778
C02413=1152.557,341.998,-78.317,-176.511,8.939,148.779
C02414=1152.553,342.245,-78.351,-176.508,8.942,148.779
C02415=1152.548,342.494,-78.385,-176.505,8.946,148.779
C02416=1152.545,342.741,-78.419,-176.503,8.950,148.779
C02417=1152.540,342.988,-78.452,-176.501,8.953,148.780
C02418=1152.536,343.236,-78.487,-176.498,8.957,148.780
C02419=1152.532,343.484,-78.520,-176.496,8.961,148.780
C02420=1152.528,343.731,-78.554,-176.493,8.965,148.780
C02421=1152.524,343.979,-78.587,-176.491,8.968,148.781
C02422=1152.520,344.227,-78.622,-176.488,8.972,148.781
C02423=1152.516,344.475,-78.655,-176.486,8.975,148.781
C02424=1152.512,344.722,-78.689,-176.483,8.980,148.782
C02425=1152.508,344.970,-78.723,-176.481,8.983,148.782
C02426=1152.504,345.217,-78.757,-176.478,8.987,148.782
C02427=1152.500,345.465,-78.791,-176.476,8.991,148.782
C02428=1152.496,345.713,-78.825,-176.473,8.995,148.783
C02429=1152.492,345.960,-78.859,-176.471,8.998,148.783
C02430=1152.489,346.208,-78.893,-176.468,9.002,148.783
C02431=1152.484,346.456,-78.927,-176.466,9.006,148.783
C02432=1152.480,346.703,-78.960,-176.463,9.010,148.784
C02433=1152.476,346.951,-78.995,-176.460,9.013,148.784
C02434=1152.472,347.199,-79.028,-176.458,9.017,148.784
C02435=1152.468,347.446,-79.062,-176.456,9.021,148.785
C02436=1152.464,347.694,-79.097,-176.453,9.025,148.785
C02437=1152.460,347.941,-79.131,-176.450,9.028,148.785
C02438=1152.455,348.189,-79.165,-176.448,9.032,148.785
C02439=1152.452,348.437,-79.199,-176.446,9.036,148.786
C02440=1152.447,348.685,-79.233,-176.443,9.040,148.786
C02441=1152.444,348.932,-79.268,-176.440,9.043,148.786
C02442=1152.440,349.180,-79.302,-176.438,9.047,148.787
C02443=1152.436,349.427,-79.336,-176.436,9.051,148.787
C02444=1152.432,349.675,-79.371,-176.433,9.055,148.787
C02445=1152.428,349.923,-79.404,-176.430,9.058,148.787
C02446=1152.423,350.170,-79.438,-176.428,9.062,148.788
C02447=1152.420,350.418,-79.473,-176.426,9.066,148.788
C02448=1152.415,350.665,-79.507,-176.423,9.070,148.788
C02449=1152.412,350.913,-79.541,-176.420,9.073,148.788
C02450=1152.408,351.161,-79.576,-176.418,9.078,148.789
C02451=1152.404,351.408,-79.610,-176.416,9.081,148.789
C02452=1152.400,351.656,-79.645,-176.413,9.085,148.789
C02453=1152.395,351.903,-79.679,-176.410,9.088,148.790
C02454=1152.392,352.151,-79.713,-176.408,9.093,148.790
C02455=1152.387,352.399,-79.748,-176.406,9.096,148.790
C02456=1152.384,352.646,-79.782,-176.403,9.100,148.790
C02457=1152.380,352.894,-79.816,-176.401,9.104,148.791
C02458=1152.376,353.142,-79.851,-176.398,9.108,148.791
C02459=1152.372,353.389,-79.885,-176.396,9.111,148.791
C02460=1152.368,353.637,-79.921,-176.393,9.115,148.792
C02461=1152.364,353.884,-79.955,-176.390,9.119,148.792
C02462=1152.360,354.132,-79.989,-176.388,9.123,148.792
C02463=1152.356,354.379,-80.024,-176.385,9.127,148.793
C02464=1152.352,354.627,-80.058,-176.383,9.130,148.793
C02465=1152.348,354.874,-80.093,-176.380,9.134,148.793
C02466=1152.344,355.122,-80.128,-176.378,9.138,148.794
C02467=1152.340,355.369,-80.162,-176.375,9.142,148.794
C02468=1152.336,355.617,-80.197,-176.373,9.145,148.794
C02469=1152.332,355.865,-80.231,-176.371,9.150,148.795
C02470=1152.328,356.113,-80.266,-176.368,9.153,148.795
C02471=1152.324,356.359,-80.301,-176.365,9.157,148.795
C02472=1152.320,356.607,-80.336,-176.363,9.162,148.795
C02473=1152.316,356.855,-80.370,-176.361,9.165,148.796
C02474=1152.312,357.102,-80.406,-176.358,9.169,148.796
C02475=1152.309,357.350,-80.440,-176.356,9.173,148.796
C02476=1152.304,357.597,-80.474,-176.353,9.177,148.797
C02477=1152.301,357.845,-80.510,-176.351,9.180,148.797
C02478=1152.296,358.092,-80.544,-176.348,9.184,148.797
C02479=1152.293,358.340,-80.579,-176.345,9.188,148.798
C02480=1152.289,358.588,-80.614,-176.343,9.192,148.798
C02481=1152.285,358.835,-80.649,-176.340,9.196,148.798
C02482=1152.281,359.083,-80.684,-176.337,9.200,148.799
C02483=1152.277,359.331,-80.719,-176.335,9.203,148.799
C02484=1152.273,359.577,-80.754,-176.333,9.208,148.799
C02485=1152.270,359.825,-80.788,-176.330,9.211,148.799
C02486=1152.265,360.072,-80.824,-176.328,9.216,148.800
C02487=1152.261,360.320,-80.858,-176.325,9.220,148.800
C02488=1152.258,360.568,-80.894,-176.323,9.223,148.800
C02489=1152.253,360.815,-80.928,-176.320,9.227,148.801
C02490=1152.249,361.063,-80.964,-176.317,9.231,148.801
C02491=1152.245,361.311,-80.999,-176.315,9.235,148.801
C02492=1152.241,361.558,-81.034,-176.312,9.239,148.802
C02493=1152.238,361.805,-81.069,-176.310,9.243,148.802
C02494=1152.234,362.053,-81.104,-176.308,9.247,148.802
C02495=1152.230,362.300,-81.139,-176.305,9.251,148.803
C02496=1152.226,362.548,-81.174,-176.302,9.255,148.803
C02497=1152.222,362.795,-81.209,-176.300,9.258,148.803
C02498=1152.218,363.042,-81.244,-176.297,9.263,148.804
C02499=1152.214,363.290,-81.279,-176.295,9.267,148.804
C02500=1152.211,363.538,-81.315,-176.292,9.270,148.804
C02501=1152.207,363.785,-81.350,-176.289,9.274,148.805
C02502=1152.203,364.032,-81.386,-176.287,9.279,148.805
C02503=1152.199,364.280,-81.420,-176.284,9.283,148.805
C02504=1152.195,364.528,-81.456,-176.282,9.286,148.806
C02505=1152.191,364.775,-81.492,-176.279,9.291,148.806
C02506=1152.186,365.058,-81.532,-176.277,9.295,148.807
C02507=1152.182,365.341,-81.573,-176.273,9.300,148.807
C02508=1152.177,365.625,-81.613,-176.271,9.304,148.807
C02509=1152.173,365.907,-81.653,-176.267,9.309,148.808
C02510=1152.169,366.154,-81.689,-176.265,9.313,148.808
C02511=1152.165,366.403,-81.724,-176.262,9.317,148.808
C02512=1152.161,366.650,-81.760,-176.260,9.321,148.809
C02513=1152.157,366.897,-81.795,-176.258,9.325,148.809
C02514=1152.153,367.145,-81.831,-176.255,9.329,148.809
C02515=1152.150,367.392,-81.866,-176.253,9.333,148.810
C02516=1152.146,367.640,-81.902,-176.250,9.337,148.810
C02517=1152.142,367.886,-81.937,-176.248,9.341,148.811
C02518=1152.137,368.134,-81.973,-176.245,9.345,148.811
C02519=1152.134,368.382,-82.009,-176.243,9.349,148.811
C02520=1152.130,368.629,-82.044,-176.241,9.353,148.812
C02521=1152.126,368.877,-82.080,-176.238,9.357,148.812
C02522=1152.123,369.124,-82.115,-176.235,9.362,148.813
C02523=1152.118,369.371,-82.151,-176.233,9.365,148.813
C02524=1152.114,369.619,-82.187,-176.231,9.370,148.813
C02525=1152.110,369.866,-82.222,-176.228,9.374,148.814
C02526=1152.107,370.114,-82.258,-176.226,9.378,148.814
C02527=1152.102,370.361,-82.294,-176.224,9.382,148.815
C02528=1152.099,370.609,-82.330,-176.221,9.386,148.815
C02529=1152.095,370.856,-82.366,-176.219,9.390,148.816
C02530=1152.091,371.103,-82.401,-176.217,9.394,148.816
C02531=1152.086,371.351,-82.437,-176.214,9.398,148.816
C02532=1152.083,371.598,-82.472,-176.212,9.402,148.817
C02533=1152.079,371.845,-82.509,-176.209,9.406,148.817
C02534=1152.075,372.093,-82.545,-176.207,9.410,148.818
C02535=1152.071,372.340,-82.580,-176.205,9.414,148.818
C02536=1152.068,372.588,-82.616,-176.203,9.418,148.818
C02537=1152.064,372.835,-82.653,-176.200,9.423,148.819
C02538=1152.060,373.083,-82.688,-176.199,9.427,148.820
C02539=1152.056,373.330,-82.724,-176.196,9.431,148.820
C02540=1152.052,373.577,-82.761,-176.194,9.435,148.820
C02541=1152.048,373.824,-82.796,-176.192,9.439,148.821
C02542=1152.044,374.072,-82.831,-176.190,9.443,148.821
C02543=1152.040,374.319,-82.868,-176.188,9.447,148.822
C02544=1152.037,374.566,-82.904,-176.186,9.451,148.822
C02545=1152.033,374.814,-82.939,-176.184,9.455,148.823
C02546=1152.029,375.061,-82.976,-176.182,9.459,148.824
C02547=1152.025,375.308,-83.012,-176.180,9.464,148.824
C02548=1152.021,375.556,-83.049,-176.178,9.468,148.825
C02549=1152.017,375.803,-83.084,-176.176,9.471,148.825
C02550=1152.013,376.051,-83.120,-176.174,9.476,148.826
C02551=1152.010,376.298,-83.157,-176.172,9.479,148.826
C02552=1152.005,376.546,-83.193,-176.170,9.484,148.827
C02553=1152.002,376.792,-83.229,-176.168,9.488,148.827
C02554=1151.997,377.040,-83.265,-176.167,9.492,148.828
C02555=1151.994,377.287,-83.301,-176.165,9.496,148.828
C02556=1151.990,377.535,-83.338,-176.163,9.500,148.829
C02557=1151.986,377.782,-83.374,-176.161,9.504,148.830
C02558=1151.982,378.030,-83.410,-176.160,9.508,148.830
C02559=1151.979,378.277,-83.446,-176.158,9.512,148.831
C02560=1151.974,378.524,-83.483,-176.157,9.516,148.831
C02561=1151.971,378.771,-83.519,-176.155,9.520,148.832
C02562=1151.967,379.018,-83.556,-176.153,9.524,148.833
C02563=1151.963,379.266,-83.591,-176.152,9.528,148.833
C02564=1151.959,379.513,-83.628,-176.151,9.532,148.834
C02565=1151.956,379.760,-83.664,-176.149,9.536,148.835
C02566=1151.951,380.008,-83.700,-176.148,9.540,148.835
C02567=1151.948,380.255,-83.737,-176.147,9.544,148.836
C02568=1151.944,380.503,-83.774,-176.146,9.547,148.837
C02569=1151.940,380.750,-83.810,-176.144,9.551,148.837
C02570=1151.937,380.997,-83.846,-176.143,9.555,148.838
C02571=1151.932,381.244,-83.883,-176.142,9.559,148.839
C02572=1151.929,381.492,-83.919,-176.141,9.563,148.839
C02573=1151.925,381.739,-83.956,-176.140,9.566,148.840
C02574=1151.921,381.986,-83.992,-176.139,9.570,148.841
C02575=1151.917,382.233,-84.029,-176.138,9.573,148.841
C02576=1151.913,382.481,-84.065,-176.137,9.578,148.842
C02577=1151.909,382.728,-84.102,-176.136,9.581,148.843
C02578=1151.905,382.975,-84.138,-176.135,9.585,148.844
C02579=1151.901,383.222,-84.175,-176.134,9.588,148.844
C02580=1151.898,383.471,-84.211,-176.133,9.593,148.845
C02581=1151.894,383.718,-84.248,-176.133,9.596,148.846
C02582=1151.890,383.965,-84.284,-176.132,9.599,148.847
C02583=1151.886,384.212,-84.321,-176.132,9.603,148.847
C02584=1151.883,384.459,-84.357,-176.131,9.607,148.848
C02585=1151.879,384.706,-84.394,-176.130,9.610,148.849
C02586=1151.874,384.954,-84.431,-176.130,9.614,148.850
C02587=1151.871,385.201,-84.467,-176.129,9.617,148.851
C02588=1151.867,385.449,-84.504,-176.129,9.620,148.851
C02589=1151.863,385.696,-84.541,-176.129,9.623,148.852
C02590=1151.860,385.943,-84.577,-176.129,9.627,148.853
C02591=1151.856,386.190,-84.614,-176.129,9.630,148.854
C02592=1151.852,386.437,-84.651,-176.128,9.633,148.854
C02593=1151.848,386.685,-84.686,-176.129,9.636,148.855
C02594=1151.844,386.932,-84.723,-176.128,9.640,148.856
C02595=1151.840,387.179,-84.760,-176.129,9.643,148.857
C02596=1151.836,387.427,-84.797,-176.128,9.646,148.858
C02597=1151.833,387.674,-84.834,-176.129,9.649,148.859
C02598=1151.829,387.921,-84.870,-176.128,9.652,148.859
C02599=1151.825,388.168,-84.907,-176.129,9.655,148.860
C02600=1151.821,388.415,-84.944,-176.129,9.658,148.861
C02601=1151.817,388.662,-84.980,-176.129,9.660,148.862
C02602=1151.814,388.910,-85.018,-176.129,9.664,148.863
C02603=1151.810,389.157,-85.054,-176.129,9.667,148.864
C02604=1151.806,389.404,-85.091,-176.130,9.670,148.864
C02605=1151.802,389.651,-85.128,-176.130,9.672,148.865
C02606=1151.798,389.899,-85.164,-176.131,9.675,148.866
C02607=1151.794,390.146,-85.201,-176.131,9.678,148.867
C02608=1151.791,390.394,-85.237,-176.132,9.681,148.868
C02609=1151.787,390.641,-85.274,-176.132,9.683,148.869
C02610=1151.783,390.927,-85.317,-176.133,9.687,148.870
C02611=1151.778,391.213,-85.359,-176.133,9.689,148.871
C02612=1151.774,391.500,-85.402,-176.134,9.692,148.871
C02613=1151.769,391.786,-85.445,-176.135,9.695,148.873
C02614=1151.765,392.034,-85.481,-176.135,9.698,148.873
C02615=1151.761,392.281,-85.518,-176.136,9.701,148.874
C02616=1151.757,392.528,-85.555,-176.137,9.703,148.875
C02617=1151.754,392.776,-85.592,-176.137,9.706,148.876
C02618=1151.750,393.023,-85.629,-176.138,9.709,148.877
C02619=1151.746,393.270,-85.666,-176.139,9.711,148.878
C02620=1151.742,393.517,-85.702,-176.139,9.714,148.879
C02621=1151.739,393.764,-85.739,-176.140,9.716,148.879
C02622=1151.735,394.012,-85.776,-176.141,9.718,148.880
C02623=1151.731,394.259,-85.813,-176.142,9.720,148.881
C02624=1151.727,394.506,-85.850,-176.142,9.723,148.882
C02625=1151.723,394.753,-85.886,-176.143,9.725,148.883
C02626=1151.720,395.000,-85.923,-176.144,9.727,148.884
C02627=1151.715,395.247,-85.960,-176.145,9.730,148.884
C02628=1151.712,395.495,-85.997,-176.146,9.732,148.885
C02629=1151.708,395.743,-86.034,-176.147,9.734,148.886
C02630=1151.704,395.990,-86.071,-176.147,9.737,148.887
C02631=1151.700,396.237,-86.107,-176.148,9.739,148.888
C02632=1151.696,396.484,-86.144,-176.149,9.741,148.888
C02633=1151.692,396.731,-86.180,-176.151,9.743,148.889
C02634=1151.689,396.979,-86.218,-176.151,9.746,148.890
C02635=1151.685,397.226,-86.255,-176.152,9.748,148.891
C02636=1151.681,397.473,-86.291,-176.153,9.750,148.892
C02637=1151.677,397.720,-86.328,-176.154,9.752,148.893
C02638=1151.673,397.967,-86.365,-176.155,9.754,148.893
C02639=1151.670,398.215,-86.402,-176.156,9.757,148.894
C02640=1151.665,398.462,-86.439,-176.156,9.759,148.895
C02641=1151.662,398.709,-86.475,-176.157,9.761,148.896
C02642=1151.658,398.957,-86.512,-176.159,9.763,148.897
C02643=1151.654,399.204,-86.549,-176.160,9.765,148.897
C02644=1151.650,399.451,-86.585,-176.161,9.767,148.898
C02645=1151.646,399.699,-86.623,-176.161,9.769,148.899
C02646=1151.643,399.946,-86.659,-176.163,9.771,148.900
C02647=1151.639,400.193,-86.696,-176.164,9.773,148.901
C02648=1151.635,400.440,-86.733,-176.164,9.774,148.901
C02649=1151.631,400.687,-86.770,-176.166,9.776,148.902
C02650=1151.627,400.935,-86.807,-176.167,9.778,148.903
C02651=1151.624,401.182,-86.843,-176.168,9.781,148.904
C02652=1151.620,401.429,-86.881,-176.168,9.782,148.904
C02653=1151.616,401.676,-86.917,-176.170,9.784,148.905
C02654=1151.612,401.923,-86.954,-176.171,9.786,148.906
C02655=1151.608,402.171,-86.992,-176.171,9.788,148.907
C02656=1151.605,402.418,-87.028,-176.172,9.790,148.908
C02657=1151.601,402.665,-87.065,-176.174,9.792,148.908
C02658=1151.597,402.912,-87.102,-176.174,9.794,148.909
C02659=1151.593,403.159,-87.138,-176.175,9.796,148.910
C02660=1151.589,403.406,-87.175,-176.176,9.798,148.911
C02661=1151.586,403.654,-87.212,-176.177,9.800,148.911
C02662=1151.582,403.901,-87.249,-176.178,9.802,148.912
C02663=1151.578,404.148,-87.286,-176.179,9.804,148.913
C02664=1151.574,404.396,-87.322,-176.180,9.806,148.914
C02665=1151.570,404.643,-87.359,-176.181,9.808,148.914
C02666=1151.566,404.891,-87.397,-176.182,9.810,148.915
C02667=1151.563,405.138,-87.433,-176.182,9.811,148.916
C02668=1151.559,405.385,-87.470,-176.184,9.813,148.917
C02669=1151.554,405.632,-87.506,-176.184,9.815,148.917
C02670=1151.550,405.879,-87.543,-176.186,9.816,148.918
C02671=1151.547,406.127,-87.581,-176.187,9.818,148.919
C02672=1151.544,406.374,-87.617,-176.187,9.820,148.919
C02673=1151.539,406.621,-87.654,-176.188,9.822,148.920
C02674=1151.535,406.868,-87.691,-176.189,9.824,148.921
C02675=1151.531,407.116,-87.727,-176.190,9.826,148.922
C02676=1151.528,407.363,-87.765,-176.191,9.828,148.922
C02677=1151.525,407.610,-87.802,-176.192,9.829,148.923
C02678=1151.521,407.857,-87.838,-176.193,9.831,148.924
C02679=1151.517,408.104,-87.875,-176.193,9.833,148.924
C02680=1151.512,408.351,-87.912,-176.194,9.835,148.925
C02681=1151.509,408.599,-87.949,-176.195,9.837,148.926
C02682=1151.505,408.846,-87.986,-176.196,9.839,148.927
C02683=1151.501,409.093,-88.023,-176.197,9.840,148.927
C02684=1151.497,409.340,-88.059,-176.198,9.842,148.928
C02685=1151.493,409.588,-88.096,-176.198,9.844,148.929
C02686=1151.490,409.835,-88.133,-176.199,9.846,148.929
C02687=1151.486,410.083,-88.170,-176.200,9.848,148.930
C02688=1151.482,410.330,-88.207,-176.201,9.850,148.931
C02689=1151.478,410.577,-88.243,-176.201,9.852,148.931
C02690=1151.474,410.824,-88.280,-176.202,9.853,148.932
C02691=1151.470,411.071,-88.317,-176.203,9.855,148.933
C02692=1151.467,411.319,-88.354,-176.204,9.857,148.934
C02693=1151.462,411.566,-88.391,-176.205,9.859,148.934
C02694=1151.459,411.813,-88.428,-176.205,9.861,148.935
C02695=1151.455,412.060,-88.464,-176.206,9.862,148.935
C02696=1151.451,412.307,-88.502,-176.207,9.864,148.936
C02697=1151.448,412.555,-88.539,-176.207,9.867,148.937
C02698=1151.444,412.802,-88.576,-176.208,9.869,148.938
C02699=1151.440,413.049,-88.613,-176.208,9.870,148.938
C02700=1151.436,413.296,-88.649,-176.209,9.872,148.939
C02701=1151.432,413.543,-88.686,-176.210,9.874,148.940
C02702=1151.429,413.791,-88.723,-176.211,9.876,148.940
C02703=1151.425,414.038,-88.760,-176.211,9.877,148.941
C02704=1151.420,414.285,-88.797,-176.212,9.879,148.941
C02705=1151.416,414.533,-88.834,-176.213,9.881,148.942
C02706=1151.413,414.780,-88.870,-176.213,9.884,148.943
C02707=1151.409,415.027,-88.907,-176.214,9.886,148.944
C02708=1151.407,415.274,-88.945,-176.214,9.887,148.944
C02709=1151.405,415.522,-88.981,-176.215,9.889,148.945
C02710=1151.405,415.738,-89.013,-176.215,9.891,148.945
C02711=1151.404,415.955,-89.045,-176.216,9.892,148.946
C02712=1151.404,416.171,-89.077,-176.216,9.894,148.946
C02713=1151.405,416.387,-89.108,-176.217,9.895,148.947
C02714=1151.407,416.604,-89.140,-176.217,9.897,148.948
C02715=1151.408,416.820,-89.172,-176.218,9.899,148.948
C02716=1151.411,417.036,-89.203,-176.218,9.900,148.949
C02717=1151.414,417.252,-89.235,-176.218,9.902,148.949
C02718=1150.994,417.253,-89.284,-176.221,9.913,148.953
C02719=1150.990,417.036,-89.252,-176.221,9.911,148.952
C02720=1150.988,416.819,-89.220,-176.221,9.909,148.952
C02721=1150.986,416.600,-89.189,-176.220,9.908,148.951
C02722=1150.984,416.382,-89.156,-176.220,9.906,148.951
C02723=1150.984,416.165,-89.125,-176.219,9.904,148.950
C02724=1150.984,415.947,-89.092,-176.219,9.903,148.950
C02725=1150.984,415.729,-89.060,-176.218,9.901,148.949
C02726=1150.984,415.510,-89.027,-176.218,9.900,148.948
C02727=1150.986,415.263,-88.991,-176.217,9.898,148.948
C02728=1150.989,415.015,-88.955,-176.216,9.896,148.947
C02729=1150.992,414.768,-88.917,-176.215,9.894,148.946
C02730=1150.996,414.521,-88.880,-176.215,9.892,148.946
C02731=1151.000,414.274,-88.843,-176.214,9.891,148.945
C02732=1151.004,414.027,-88.807,-176.214,9.888,148.944
C02733=1151.007,413.779,-88.769,-176.213,9.886,148.944
C02734=1151.011,413.532,-88.733,-176.212,9.885,148.943
C02735=1151.016,413.285,-88.696,-176.212,9.883,148.942
C02736=1151.019,413.038,-88.659,-176.211,9.881,148.942
C02737=1151.023,412.791,-88.623,-176.210,9.879,148.941
C02738=1151.027,412.543,-88.585,-176.209,9.877,148.940
C02739=1151.031,412.295,-88.548,-176.209,9.876,148.940
C02740=1151.034,412.049,-88.511,-176.208,9.874,148.939
C02741=1151.039,411.802,-88.474,-176.207,9.872,148.938
C02742=1151.043,411.555,-88.437,-176.206,9.870,148.938
C02743=1151.045,411.307,-88.401,-176.206,9.867,148.937
C02744=1151.049,411.060,-88.364,-176.205,9.866,148.936
C02745=1151.054,410.813,-88.327,-176.205,9.864,148.936
C02746=1151.058,410.565,-88.290,-176.204,9.862,148.935
C02747=1151.062,410.318,-88.253,-176.203,9.860,148.934
C02748=1151.065,410.070,-88.216,-176.202,9.858,148.933
C02749=1151.069,409.823,-88.180,-176.202,9.857,148.933
C02750=1151.073,409.576,-88.143,-176.201,9.855,148.932
C02751=1151.077,409.329,-88.106,-176.200,9.853,148.931
C02752=1151.081,409.082,-88.069,-176.199,9.851,148.931
C02753=1151.084,408.834,-88.032,-176.198,9.849,148.930
C02754=1151.088,408.587,-87.996,-176.197,9.847,148.929
C02755=1151.092,408.341,-87.958,-176.197,9.846,148.929
C02756=1151.096,408.093,-87.921,-176.196,9.843,148.928
C02757=1151.100,407.846,-87.884,-176.195,9.842,148.927
C02758=1151.103,407.598,-87.847,-176.194,9.840,148.926
C02759=1151.107,407.351,-87.810,-176.193,9.839,148.926
C02760=1151.111,407.104,-87.774,-176.192,9.837,148.925
C02761=1151.115,406.857,-87.737,-176.191,9.835,148.924
C02762=1151.119,406.610,-87.700,-176.190,9.833,148.924
C02763=1151.122,406.362,-87.663,-176.189,9.831,148.923
C02764=1151.126,406.115,-87.626,-176.188,9.829,148.922
C02765=1151.130,405.868,-87.590,-176.188,9.828,148.921
C02766=1151.134,405.621,-87.553,-176.187,9.826,148.921
C02767=1151.138,405.373,-87.516,-176.186,9.824,148.920
C02768=1151.141,405.126,-87.479,-176.185,9.822,148.919
C02769=1151.146,404.878,-87.442,-176.184,9.820,148.918
C02770=1151.150,404.631,-87.405,-176.183,9.818,148.918
C02771=1151.153,404.384,-87.369,-176.182,9.816,148.917
C02772=1151.157,404.138,-87.331,-176.181,9.814,148.916
C02773=1151.160,403.890,-87.294,-176.180,9.812,148.915
C02774=1151.164,403.643,-87.257,-176.179,9.810,148.915
C02775=1151.168,403.395,-87.220,-176.178,9.808,148.914
C02776=1151.172,403.149,-87.184,-176.178,9.806,148.913
C02777=1151.176,402.901,-87.147,-176.176,9.805,148.912
C02778=1151.180,402.654,-87.110,-176.175,9.803,148.912
C02779=1151.184,402.406,-87.073,-176.174,9.801,148.911
C02780=1151.188,402.159,-87.036,-176.173,9.799,148.910
C02781=1151.192,401.912,-87.000,-176.172,9.797,148.909
C02782=1151.195,401.665,-86.963,-176.171,9.796,148.909
C02783=1151.199,401.418,-86.926,-176.170,9.793,148.908
C02784=1151.203,401.170,-86.889,-176.169,9.791,148.907
C02785=1151.207,400.923,-86.852,-176.168,9.790,148.906
C02786=1151.211,400.676,-86.815,-176.167,9.788,148.905
C02787=1151.214,400.429,-86.779,-176.166,9.786,148.905
C02788=1151.218,400.182,-86.742,-176.165,9.783,148.904
C02789=1151.222,399.934,-86.705,-176.164,9.782,148.903
C02790=1151.226,399.686,-86.668,-176.163,9.780,148.902
C02791=1151.230,399.439,-86.631,-176.162,9.778,148.901
C02792=1151.234,399.192,-86.595,-176.161,9.776,148.901
C02793=1151.237,398.945,-86.558,-176.161,9.773,148.900
C02794=1151.241,398.698,-86.520,-176.160,9.771,148.899
C02795=1151.245,398.451,-86.483,-176.159,9.769,148.898
C02796=1151.249,398.204,-86.447,-176.158,9.767,148.897
C02797=1151.253,397.956,-86.410,-176.156,9.765,148.897
C02798=1151.256,397.709,-86.373,-176.156,9.763,148.896
C02799=1151.260,397.462,-86.336,-176.155,9.761,148.895
C02800=1151.264,397.214,-86.299,-176.153,9.759,148.894
C02801=1151.268,396.967,-86.263,-176.153,9.756,148.893
C02802=1151.272,396.720,-86.226,-176.152,9.754,148.892
C02803=1151.275,396.473,-86.189,-176.151,9.752,148.892
C02804=1151.279,396.226,-86.153,-176.150,9.750,148.891
C02805=1151.283,395.978,-86.115,-176.150,9.747,148.890
C02806=1151.287,395.731,-86.078,-176.148,9.745,148.889
C02807=1151.291,395.484,-86.042,-176.147,9.743,148.888
C02808=1151.295,395.237,-86.005,-176.146,9.741,148.888
C02809=1151.299,394.990,-85.969,-176.146,9.738,148.887
C02810=1151.302,394.742,-85.931,-176.145,9.736,148.886
C02811=1151.306,394.494,-85.894,-176.144,9.733,148.885
C02812=1151.310,394.247,-85.858,-176.143,9.732,148.884
C02813=1151.314,394.000,-85.821,-176.142,9.729,148.883
C02814=1151.318,393.753,-85.784,-176.142,9.727,148.883
C02815=1151.322,393.506,-85.748,-176.141,9.725,148.882
C02816=1151.325,393.258,-85.710,-176.140,9.722,148.881
C02817=1151.329,393.011,-85.674,-176.139,9.720,148.880
C02818=1151.333,392.764,-85.637,-176.138,9.717,148.879
C02819=1151.337,392.517,-85.600,-176.138,9.714,148.878
C02820=1151.341,392.270,-85.564,-176.137,9.712,148.878
C02821=1151.344,392.022,-85.526,-176.137,9.709,148.877
C02822=1151.348,391.775,-85.490,-176.136,9.706,148.876
C02823=1151.353,391.488,-85.446,-176.136,9.703,148.875
C02824=1151.358,391.202,-85.404,-176.135,9.700,148.874
C02825=1151.362,390.916,-85.362,-176.134,9.697,148.873
C02826=1151.366,390.629,-85.319,-176.134,9.695,148.872
C02827=1151.370,390.383,-85.283,-176.133,9.692,148.871
C02828=1151.374,390.135,-85.246,-176.132,9.689,148.870
C02829=1151.377,389.888,-85.209,-176.132,9.686,148.869
C02830=1151.381,389.640,-85.172,-176.132,9.683,148.869
C02831=1151.385,389.393,-85.135,-176.131,9.681,148.868
C02832=1151.389,389.146,-85.099,-176.131,9.678,148.867
C02833=1151.393,388.899,-85.062,-176.131,9.675,148.866
C02834=1151.397,388.652,-85.025,-176.130,9.672,148.865
C02835=1151.400,388.404,-84.988,-176.130,9.669,148.864
C02836=1151.404,388.156,-84.952,-176.130,9.666,148.864
C02837=1151.408,387.909,-84.915,-176.130,9.663,148.863
C02838=1151.412,387.662,-84.878,-176.130,9.660,148.862
C02839=1151.416,387.415,-84.842,-176.129,9.657,148.861
C02840=1151.420,387.168,-84.805,-176.129,9.654,148.860
C02841=1151.423,386.920,-84.768,-176.129,9.651,148.859
C02842=1151.427,386.673,-84.731,-176.130,9.647,148.859
C02843=1151.431,386.426,-84.695,-176.130,9.645,148.858
C02844=1151.435,386.179,-84.658,-176.130,9.641,148.857
C02845=1151.439,385.932,-84.621,-176.130,9.638,148.856
C02846=1151.442,385.685,-84.585,-176.130,9.635,148.855
C02847=1151.447,385.437,-84.549,-176.131,9.632,148.855
C02848=1151.450,385.189,-84.512,-176.131,9.628,148.854
C02849=1151.453,384.942,-84.475,-176.131,9.625,148.853
C02850=1151.457,384.695,-84.438,-176.132,9.621,148.852
C02851=1151.462,384.448,-84.402,-176.132,9.618,148.851
C02852=1151.466,384.201,-84.365,-176.133,9.614,148.851
C02853=1151.469,383.954,-84.329,-176.134,9.610,148.850
C02854=1151.473,383.706,-84.292,-176.134,9.607,148.849
C02855=1151.478,383.459,-84.256,-176.135,9.603,148.848
C02856=1151.480,383.211,-84.219,-176.135,9.600,148.848
C02857=1151.484,382.964,-84.182,-176.137,9.596,148.847
C02858=1151.488,382.717,-84.145,-176.137,9.593,148.846
C02859=1151.492,382.469,-84.110,-176.138,9.589,148.845
C02860=1151.496,382.222,-84.073,-176.139,9.585,148.845
C02861=1151.500,381.975,-84.036,-176.140,9.581,148.844
C02862=1151.504,381.728,-84.000,-176.141,9.577,148.843
C02863=1151.508,381.480,-83.963,-176.142,9.574,148.843
C02864=1151.511,381.233,-83.927,-176.143,9.570,148.842
C02865=1151.516,380.986,-83.890,-176.144,9.566,148.841
C02866=1151.520,380.739,-83.854,-176.146,9.562,148.841
C02867=1151.523,380.491,-83.818,-176.147,9.559,148.840
C02868=1151.527,380.244,-83.781,-176.148,9.555,148.839
C02869=1151.530,379.997,-83.744,-176.149,9.551,148.839
C02870=1151.535,379.749,-83.708,-176.151,9.547,148.838
C02871=1151.538,379.502,-83.672,-176.152,9.543,148.837
C02872=1151.542,379.255,-83.635,-176.154,9.539,148.837
C02873=1151.546,379.007,-83.599,-176.155,9.535,148.836
C02874=1151.550,378.760,-83.563,-176.157,9.531,148.836
C02875=1151.554,378.512,-83.527,-176.158,9.528,148.835
C02876=1151.557,378.265,-83.490,-176.160,9.523,148.834
C02877=1151.562,378.018,-83.454,-176.162,9.519,148.834
C02878=1151.565,377.771,-83.418,-176.163,9.515,148.833
C02879=1151.569,377.524,-83.381,-176.165,9.511,148.832
C02880=1151.573,377.276,-83.346,-176.167,9.506,148.832
C02881=1151.577,377.029,-83.309,-176.169,9.503,148.831
C02882=1151.581,376.781,-83.273,-176.170,9.499,148.831
C02883=1151.585,376.534,-83.236,-176.172,9.495,148.830
C02884=1151.589,376.287,-83.201,-176.174,9.491,148.830
C02885=1151.593,376.040,-83.164,-176.176,9.487,148.829
C02886=1151.596,375.792,-83.128,-176.178,9.482,148.828
C02887=1151.600,375.545,-83.092,-176.179,9.478,148.828
C02888=1151.604,375.297,-83.056,-176.181,9.475,148.827
C02889=1151.608,375.049,-83.020,-176.184,9.471,148.827
C02890=1151.612,374.803,-82.984,-176.185,9.467,148.826
C02891=1151.615,374.555,-82.948,-176.188,9.462,148.826
C02892=1151.620,374.308,-82.911,-176.190,9.459,148.825
C02893=1151.623,374.060,-82.876,-176.192,9.454,148.825
C02894=1151.628,373.813,-82.839,-176.194,9.450,148.824
C02895=1151.631,373.566,-82.803,-176.196,9.446,148.824
C02896=1151.635,373.318,-82.768,-176.199,9.442,148.823
C02897=1151.639,373.070,-82.732,-176.200,9.438,148.823
C02898=1151.643,372.824,-82.696,-176.203,9.433,148.822
C02899=1151.647,372.577,-82.660,-176.204,9.430,148.822
C02900=1151.651,372.329,-82.624,-176.207,9.425,148.821
C02901=1151.655,372.081,-82.588,-176.209,9.421,148.821
C02902=1151.658,371.835,-82.552,-176.211,9.417,148.821
C02903=1151.662,371.587,-82.516,-176.214,9.413,148.820
C02904=1151.666,371.339,-82.480,-176.217,9.409,148.820
C02905=1151.670,371.092,-82.445,-176.219,9.405,148.819
C02906=1151.673,370.845,-82.409,-176.221,9.401,148.819
C02907=1151.678,370.597,-82.372,-176.224,9.396,148.818
C02908=1151.682,370.350,-82.337,-176.225,9.393,148.818
C02909=1151.685,370.103,-82.302,-176.228,9.388,148.818
C02910=1151.690,369.855,-82.266,-176.230,9.384,148.817
C02911=1151.694,369.607,-82.230,-176.233,9.381,148.817
C02912=1151.697,369.360,-82.194,-176.235,9.376,148.816
C02913=1151.701,369.112,-82.159,-176.238,9.372,148.816
C02914=1151.705,368.865,-82.123,-176.240,9.369,148.816
C02915=1151.710,368.618,-82.088,-176.242,9.364,148.815
C02916=1151.713,368.371,-82.051,-176.245,9.360,148.815
C02917=1151.717,368.123,-82.016,-176.248,9.356,148.814
C02918=1151.720,367.876,-81.980,-176.250,9.352,148.814
C02919=1151.724,367.628,-81.945,-176.252,9.348,148.814
C02920=1151.729,367.381,-81.910,-176.255,9.344,148.813
C02921=1151.733,367.133,-81.874,-176.257,9.340,148.813
C02922=1151.737,366.886,-81.839,-176.260,9.336,148.813
C02923=1151.740,366.638,-81.803,-176.262,9.332,148.812
C02924=1151.744,366.391,-81.767,-176.265,9.328,148.812
C02925=1151.748,366.144,-81.732,-176.267,9.324,148.811
C02926=1151.752,365.896,-81.697,-176.270,9.320,148.811
C02927=1151.756,365.613,-81.656,-176.273,9.315,148.811
C02928=1151.761,365.330,-81.615,-176.276,9.310,148.810
C02929=1151.766,365.047,-81.575,-176.279,9.306,148.810
C02930=1151.769,364.764,-81.535,-176.282,9.301,148.809
C02931=1151.773,364.516,-81.499,-176.284,9.298,148.809
C02932=1151.778,364.269,-81.465,-176.286,9.293,148.809
C02933=1151.781,364.022,-81.429,-176.289,9.289,148.808
C02934=1151.785,363.774,-81.393,-176.292,9.285,148.808
C02935=1151.789,363.527,-81.358,-176.294,9.282,148.808
C02936=1151.793,363.279,-81.323,-176.297,9.277,148.808
C02937=1151.797,363.032,-81.288,-176.300,9.273,148.807
C02938=1151.800,362.784,-81.252,-176.302,9.270,148.807
C02939=1151.805,362.537,-81.218,-176.305,9.266,148.807
C02940=1151.809,362.289,-81.182,-176.307,9.261,148.806
C02941=1151.812,362.042,-81.147,-176.310,9.258,148.806
C02942=1151.816,361.794,-81.112,-176.312,9.254,148.805
C02943=1151.821,361.547,-81.077,-176.315,9.249,148.805
C02944=1151.824,361.299,-81.041,-176.318,9.245,148.805
C02945=1151.828,361.051,-81.006,-176.320,9.242,148.804
C02946=1151.832,360.804,-80.971,-176.323,9.238,148.804
C02947=1151.836,360.556,-80.936,-176.326,9.234,148.804
C02948=1151.840,360.309,-80.901,-176.327,9.230,148.804
C02949=1151.845,360.061,-80.866,-176.330,9.226,148.803
C02950=1151.848,359.814,-80.831,-176.332,9.222,148.803
C02951=1151.852,359.567,-80.797,-176.335,9.218,148.803
C02952=1151.856,359.319,-80.761,-176.338,9.214,148.802
C02953=1151.860,359.071,-80.727,-176.340,9.211,148.802
C02954=1151.864,358.824,-80.691,-176.343,9.206,148.802
C02955=1151.868,358.576,-80.657,-176.346,9.202,148.801
C02956=1151.871,358.329,-80.622,-176.348,9.199,148.801
C02957=1151.875,358.082,-80.587,-176.351,9.195,148.801
C02958=1151.879,357.833,-80.552,-176.353,9.191,148.800
C02959=1151.884,357.587,-80.517,-176.355,9.187,148.800
C02960=1151.888,357.339,-80.482,-176.358,9.183,148.800
C02961=1151.892,357.091,-80.448,-176.360,9.179,148.799
C02962=1151.895,356.844,-80.413,-176.363,9.175,148.799
C02963=1151.899,356.596,-80.378,-176.365,9.172,148.799
C02964=1151.904,356.348,-80.344,-176.368,9.168,148.798
C02965=1151.907,356.101,-80.309,-176.370,9.164,148.798
C02966=1151.911,355.854,-80.274,-176.373,9.160,148.798
C02967=1151.915,355.606,-80.239,-176.376,9.156,148.797
C02968=1151.920,355.358,-80.205,-176.378,9.153,148.797
C02969=1151.923,355.111,-80.170,-176.381,9.148,148.797
C02970=1151.927,354.864,-80.135,-176.383,9.145,148.797
C02971=1151.931,354.615,-80.101,-176.386,9.141,148.796
C02972=1151.935,354.368,-80.067,-176.388,9.138,148.796
C02973=1151.939,354.120,-80.032,-176.390,9.133,148.796
C02974=1151.943,353.873,-79.997,-176.393,9.130,148.795
C02975=1151.947,353.626,-79.962,-176.396,9.126,148.795
C02976=1151.951,353.378,-79.928,-176.398,9.121,148.795
C02977=1151.955,353.130,-79.893,-176.400,9.118,148.794
C02978=1151.959,352.883,-79.859,-176.403,9.114,148.794
C02979=1151.963,352.635,-79.824,-176.405,9.110,148.794
C02980=1151.967,352.388,-79.791,-176.408,9.106,148.794
C02981=1151.971,352.140,-79.756,-176.410,9.103,148.793
C02982=1151.975,351.892,-79.721,-176.413,9.099,148.793
C02983=1151.978,351.644,-79.687,-176.415,9.095,148.793
C02984=1151.983,351.397,-79.653,-176.418,9.091,148.792
C02985=1151.986,351.149,-79.618,-176.420,9.088,148.792
C02986=1151.991,350.902,-79.584,-176.423,9.084,148.792
C02987=1151.995,350.655,-79.550,-176.425,9.080,148.792
C02988=1151.999,350.407,-79.515,-176.428,9.076,148.791
C02989=1152.002,350.159,-79.481,-176.430,9.073,148.791
C02990=1152.006,349.911,-79.446,-176.433,9.069,148.791
C02991=1152.011,349.664,-79.412,-176.436,9.064,148.790
C02992=1152.015,349.417,-79.378,-176.438,9.061,148.790
C02993=1152.019,349.169,-79.343,-176.441,9.057,148.790
C02994=1152.023,348.922,-79.309,-176.443,9.053,148.789
C02995=1152.026,348.673,-79.276,-176.446,9.049,148.789
C02996=1152.031,348.426,-79.241,-176.448,9.046,148.789
C02997=1152.035,348.179,-79.208,-176.451,9.042,148.789
C02998=1152.039,347.930,-79.173,-176.453,9.038,148.788
C02999=1152.042,347.683,-79.139,-176.456,9.034,148.788
C03000=1152.047,347.435,-79.105,-176.458,9.031,148.788
C03001=1152.050,347.188,-79.071,-176.461,9.027,148.788
C03002=1152.055,346.940,-79.036,-176.463,9.023,148.787
C03003=1152.059,346.693,-79.003,-176.466,9.019,148.787
C03004=1152.062,346.445,-78.969,-176.468,9.016,148.787
C03005=1152.067,346.197,-78.935,-176.471,9.012,148.787
C03006=1152.071,345.950,-78.901,-176.473,9.009,148.786
C03007=1152.075,345.701,-78.867,-176.476,9.004,148.786
C03008=1152.079,345.454,-78.833,-176.478,9.001,148.786
C03009=1152.083,345.207,-78.799,-176.481,8.997,148.785
C03010=1152.087,344.958,-78.765,-176.483,8.994,148.785
C03011=1152.091,344.711,-78.731,-176.486,8.990,148.785
C03012=1152.095,344.463,-78.698,-176.488,8.986,148.785
C03013=1152.099,344.215,-78.663,-176.490,8.983,148.784
C03014=1152.103,343.968,-78.629,-176.493,8.979,148.784
C03015=1152.107,343.721,-78.596,-176.496,8.975,148.784
C03016=1152.112,343.473,-78.561,-176.499,8.971,148.784
C03017=1152.115,343.225,-78.528,-176.500,8.968,148.783
C03018=1152.119,342.978,-78.494,-176.503,8.964,148.783
C03019=1152.123,342.730,-78.461,-176.506,8.960,148.783
C03020=1152.128,342.482,-78.426,-176.509,8.956,148.783
C03021=1152.131,342.234,-78.393,-176.511,8.953,148.782
C03022=1152.135,341.987,-78.359,-176.514,8.949,148.782
C03023=1152.139,341.739,-78.326,-176.516,8.945,148.782
C03024=1152.144,341.491,-78.292,-176.519,8.941,148.781
C03025=1152.148,341.244,-78.258,-176.521,8.938,148.781
C03026=1152.151,340.996,-78.225,-176.524,8.934,148.781
C03027=1152.155,340.748,-78.191,-176.526,8.930,148.781
C03028=1152.159,340.501,-78.158,-176.528,8.927,148.781
C03029=1152.164,340.253,-78.124,-176.531,8.923,148.780
C03030=1152.168,340.006,-78.090,-176.534,8.920,148.780
C03031=1152.172,339.725,-78.052,-176.536,8.915,148.780
C03032=1152.177,339.445,-78.014,-176.539,8.911,148.779
C03033=1152.182,339.164,-77.977,-176.542,8.907,148.779
C03034=1152.186,338.885,-77.939,-176.545,8.903,148.779
C03035=1152.189,338.637,-77.905,-176.548,8.899,148.779
C03036=1152.194,338.389,-77.872,-176.550,8.896,148.778
C03037=1152.199,338.141,-77.838,-176.553,8.892,148.778
C03038=1152.203,337.894,-77.805,-176.555,8.888,148.778
C03039=1152.206,337.646,-77.771,-176.558,8.884,148.778
C03040=1152.211,337.399,-77.738,-176.560,8.881,148.777
C03041=1152.215,337.151,-77.705,-176.562,8.877,148.777
C03042=1152.218,336.903,-77.671,-176.565,8.873,148.777
C03043=1152.222,336.655,-77.638,-176.568,8.870,148.777
C03044=1152.227,336.407,-77.605,-176.570,8.866,148.776
C03045=1152.231,336.159,-77.572,-176.573,8.863,148.776
C03046=1152.235,335.912,-77.538,-176.576,8.859,148.776
C03047=1152.239,335.665,-77.505,-176.578,8.855,148.776
C03048=1152.243,335.417,-77.472,-176.580,8.852,148.776
C03049=1152.247,335.169,-77.438,-176.583,8.848,148.775
C03050=1152.251,334.921,-77.405,-176.586,8.845,148.775
C03051=1152.255,334.673,-77.372,-176.588,8.841,148.775
C03052=1152.259,334.425,-77.339,-176.591,8.837,148.775
C03053=1152.263,334.177,-77.305,-176.593,8.834,148.775
C03054=1152.267,333.930,-77.272,-176.596,8.830,148.774
C03055=1152.271,333.682,-77.239,-176.598,8.827,148.774
C03056=1152.275,333.434,-77.206,-176.601,8.822,148.774
C03057=1152.279,333.187,-77.173,-176.603,8.819,148.773
C03058=1152.283,332.939,-77.140,-176.605,8.816,148.773
C03059=1152.287,332.691,-77.108,-176.608,8.812,148.773
C03060=1152.291,332.443,-77.075,-176.611,8.808,148.773
C03061=1152.296,332.195,-77.042,-176.614,8.804,148.773
C03062=1152.300,331.948,-77.008,-176.616,8.801,148.772
C03063=1152.304,331.700,-76.975,-176.618,8.798,148.772
C03064=1152.308,331.452,-76.942,-176.621,8.794,148.772
C03065=1152.311,331.205,-76.910,-176.623,8.790,148.772
C03066=1152.316,330.956,-76.877,-176.626,8.786,148.771
C03067=1152.320,330.709,-76.844,-176.629,8.783,148.771
C03068=1152.324,330.461,-76.811,-176.631,8.780,148.771
C03069=1152.328,330.213,-76.778,-176.634,8.776,148.771
C03070=1152.332,329.966,-76.745,-176.636,8.772,148.771
C03071=1152.336,329.717,-76.713,-176.638,8.769,148.770
C03072=1152.340,329.470,-76.679,-176.641,8.765,148.770
C03073=1152.344,329.222,-76.646,-176.644,8.762,148.770
C03074=1152.349,328.974,-76.614,-176.647,8.758,148.770
C03075=1152.352,328.726,-76.581,-176.649,8.755,148.770
C03076=1152.356,328.478,-76.548,-176.652,8.751,148.770
C03077=1152.361,328.230,-76.516,-176.655,8.747,148.769
C03078=1152.365,327.982,-76.483,-176.657,8.744,148.769
C03079=1152.369,327.736,-76.450,-176.659,8.741,148.769
C03080=1152.373,327.487,-76.418,-176.662,8.737,148.769
C03081=1152.378,327.240,-76.385,-176.664,8.733,148.769
C03082=1152.381,326.992,-76.353,-176.667,8.729,148.768
C03083=1152.385,326.744,-76.320,-176.670,8.726,148.768
C03084=1152.389,326.496,-76.287,-176.672,8.723,148.768
C03085=1152.393,326.248,-76.255,-176.675,8.719,148.768
C03086=1152.397,326.000,-76.222,-176.677,8.715,148.767
C03087=1152.402,325.752,-76.189,-176.679,8.712,148.767
C03088=1152.405,325.505,-76.157,-176.682,8.708,148.767
C03089=1152.410,325.257,-76.125,-176.685,8.705,148.767
C03090=1152.414,325.009,-76.091,-176.687,8.702,148.767
C03091=1152.418,324.761,-76.060,-176.690,8.698,148.767
C03092=1152.423,324.513,-76.027,-176.693,8.694,148.766
C03093=1152.426,324.265,-75.995,-176.695,8.691,148.766
C03094=1152.430,324.017,-75.962,-176.698,8.687,148.766
C03095=1152.434,323.770,-75.930,-176.700,8.684,148.766
C03096=1152.439,323.522,-75.897,-176.703,8.680,148.766
C03097=1152.443,323.274,-75.865,-176.705,8.676,148.765
C03098=1152.447,323.026,-75.832,-176.708,8.673,148.765
C03099=1152.451,322.778,-75.800,-176.710,8.670,148.765
C03100=1152.454,322.530,-75.767,-176.713,8.666,148.765
C03101=1152.459,322.282,-75.735,-176.716,8.663,148.765
C03102=1152.463,322.035,-75.704,-176.718,8.659,148.765
C03103=1152.468,321.786,-75.671,-176.721,8.655,148.764
C03104=1152.471,321.539,-75.639,-176.723,8.652,148.764
C03105=1152.476,321.291,-75.606,-176.726,8.649,148.764
C03106=1152.479,321.043,-75.574,-176.729,8.645,148.764
C03107=1152.484,320.795,-75.542,-176.731,8.642,148.764
C03108=1152.488,320.548,-75.510,-176.734,8.639,148.764
C03109=1152.491,320.299,-75.478,-176.736,8.634,148.763
C03110=1152.496,320.051,-75.445,-176.739,8.631,148.763
C03111=1152.500,319.804,-75.414,-176.741,8.628,148.763
C03112=1152.505,319.555,-75.381,-176.744,8.624,148.763
C03113=1152.508,319.307,-75.350,-176.747,8.621,148.763
C03114=1152.512,319.060,-75.317,-176.749,8.618,148.763
C03115=1152.517,318.812,-75.285,-176.751,8.614,148.762
C03116=1152.520,318.564,-75.253,-176.754,8.610,148.762
C03117=1152.525,318.316,-75.221,-176.757,8.607,148.762
C03118=1152.529,318.068,-75.189,-176.759,8.604,148.762
C03119=1152.533,317.821,-75.157,-176.762,8.600,148.762
C03120=1152.537,317.572,-75.125,-176.765,8.597,148.762
C03121=1152.541,317.324,-75.093,-176.767,8.593,148.761
C03122=1152.545,317.077,-75.062,-176.770,8.589,148.761
C03123=1152.550,316.828,-75.029,-176.773,8.586,148.761
C03124=1152.554,316.580,-74.997,-176.775,8.583,148.761
C03125=1152.558,316.333,-74.966,-176.777,8.580,148.761
C03126=1152.562,316.085,-74.933,-176.780,8.576,148.760
C03127=1152.566,315.837,-74.901,-176.782,8.572,148.760
C03128=1152.570,315.589,-74.870,-176.785,8.569,148.760
C03129=1152.574,315.341,-74.838,-176.788,8.565,148.760
C03130=1152.578,315.093,-74.806,-176.790,8.562,148.760
C03131=1152.583,314.846,-74.774,-176.793,8.559,148.760
C03132=1152.587,314.597,-74.743,-176.795,8.556,148.760
C03133=1152.590,314.349,-74.711,-176.798,8.552,148.760
C03134=1152.595,314.101,-74.679,-176.801,8.548,148.759
C03135=1152.600,313.824,-74.644,-176.804,8.544,148.759
C03136=1152.604,313.546,-74.608,-176.807,8.541,148.759
C03137=1152.609,313.269,-74.573,-176.809,8.537,148.759
C03138=1152.614,312.991,-74.538,-176.812,8.533,148.759
C03139=1152.617,312.743,-74.506,-176.814,8.530,148.758
C03140=1152.622,312.496,-74.475,-176.818,8.526,148.758
C03141=1152.626,312.248,-74.442,-176.820,8.523,148.758
C03142=1152.630,311.999,-74.411,-176.822,8.520,148.758
C03143=1152.634,311.752,-74.379,-176.825,8.517,148.758
C03144=1152.638,311.504,-74.348,-176.828,8.513,148.758
C03145=1152.642,311.256,-74.316,-176.830,8.509,148.758
C03146=1152.646,311.008,-74.285,-176.833,8.506,148.758
C03147=1152.651,310.760,-74.254,-176.835,8.503,148.758
C03148=1152.655,310.512,-74.221,-176.838,8.499,148.757
C03149=1152.660,310.264,-74.190,-176.841,8.496,148.757
C03150=1152.664,310.016,-74.158,-176.843,8.493,148.757
C03151=1152.668,309.767,-74.127,-176.846,8.489,148.757
C03152=1152.672,309.520,-74.096,-176.849,8.485,148.757
C03153=1152.676,309.272,-74.064,-176.851,8.482,148.757
C03154=1152.680,309.024,-74.033,-176.854,8.479,148.757
C03155=1152.684,308.776,-74.001,-176.856,8.476,148.756
C03156=1152.689,308.528,-73.971,-176.859,8.472,148.756
C03157=1152.692,308.280,-73.939,-176.862,8.469,148.756
C03158=1152.697,308.032,-73.908,-176.864,8.466,148.756
C03159=1152.701,307.784,-73.876,-176.867,8.463,148.756
C03160=1152.705,307.536,-73.845,-176.870,8.458,148.756
C03161=1152.709,307.288,-73.814,-176.872,8.455,148.756
C03162=1152.713,307.040,-73.783,-176.875,8.452,148.756
C03163=1152.718,306.792,-73.752,-176.877,8.449,148.755
C03164=1152.722,306.544,-73.720,-176.880,8.445,148.755
C03165=1152.726,306.296,-73.689,-176.883,8.442,148.755
C03166=1152.730,306.048,-73.658,-176.885,8.439,148.755
C03167=1152.735,305.800,-73.627,-176.887,8.435,148.755
C03168=1152.739,305.551,-73.596,-176.890,8.432,148.755
C03169=1152.743,305.304,-73.564,-176.893,8.428,148.755
C03170=1152.747,305.055,-73.533,-176.895,8.425,148.755
C03171=1152.751,304.808,-73.503,-176.898,8.422,148.755
C03172=1152.755,304.560,-73.471,-176.900,8.419,148.754
C03173=1152.759,304.312,-73.440,-176.904,8.415,148.754
C03174=1152.764,304.064,-73.410,-176.906,8.412,148.754
C03175=1152.768,303.815,-73.378,-176.908,8.409,148.754
C03176=1152.772,303.568,-73.347,-176.911,8.406,148.754
C03177=1152.777,303.320,-73.316,-176.913,8.402,148.754
C03178=1152.781,303.071,-73.285,-176.917,8.399,148.754
C03179=1152.785,302.823,-73.255,-176.919,8.395,148.754
C03180=1152.789,302.576,-73.223,-176.921,8.392,148.753
C03181=1152.793,302.327,-73.192,-176.924,8.389,148.754
C03182=1152.798,302.079,-73.162,-176.927,8.386,148.753
C03183=1152.802,301.831,-73.130,-176.930,8.382,148.753
C03184=1152.806,301.583,-73.100,-176.932,8.379,148.753
C03185=1152.810,301.335,-73.069,-176.934,8.375,148.753
C03186=1152.814,301.086,-73.038,-176.937,8.372,148.753
C03187=1152.819,300.839,-73.008,-176.940,8.369,148.753
C03188=1152.823,300.591,-72.976,-176.943,8.365,148.753
C03189=1152.826,300.343,-72.946,-176.945,8.362,148.753
C03190=1152.831,300.095,-72.915,-176.948,8.359,148.753
C03191=1152.836,299.847,-72.884,-176.950,8.356,148.752
C03192=1152.839,299.599,-72.853,-176.953,8.353,148.752
C03193=1152.843,299.351,-72.823,-176.956,8.349,148.752
C03194=1152.848,299.103,-72.792,-176.958,8.346,148.752
C03195=1152.852,298.855,-72.762,-176.961,8.343,148.752
C03196=1152.856,298.606,-72.731,-176.963,8.339,148.752
C03197=1152.861,298.358,-72.700,-176.966,8.336,148.752
C03198=1152.864,298.111,-72.670,-176.968,8.333,148.752
C03199=1152.869,297.861,-72.639,-176.972,8.329,148.752
C03200=1152.873,297.614,-72.609,-176.974,8.326,148.752
C03201=1152.877,297.366,-72.578,-176.977,8.323,148.752
C03202=1152.882,297.118,-72.548,-176.979,8.320,148.752
C03203=1152.886,296.869,-72.516,-176.982,8.317,148.752
C03204=1152.890,296.622,-72.486,-176.985,8.313,148.751
C03205=1152.894,296.374,-72.456,-176.988,8.310,148.751
C03206=1152.898,296.126,-72.425,-176.990,8.307,148.751
C03207=1152.903,295.877,-72.395,-176.993,8.304,148.751
C03208=1152.907,295.629,-72.364,-176.995,8.300,148.751
C03209=1152.911,295.381,-72.334,-176.998,8.297,148.751
C03210=1152.916,295.133,-72.303,-177.000,8.294,148.751
C03211=1152.920,294.886,-72.273,-177.003,8.290,148.751
C03212=1152.924,294.636,-72.243,-177.006,8.287,148.751
C03213=1152.928,294.389,-72.213,-177.009,8.284,148.751
C03214=1152.932,294.141,-72.182,-177.011,8.281,148.751
C03215=1152.937,293.892,-72.152,-177.014,8.278,148.751
C03216=1152.941,293.644,-72.122,-177.016,8.275,148.750
C03217=1152.944,293.396,-72.091,-177.019,8.271,148.750
C03218=1152.949,293.148,-72.060,-177.022,8.268,148.750
C03219=1152.953,292.900,-72.031,-177.024,8.265,148.750
C03220=1152.958,292.652,-72.000,-177.027,8.261,148.750
C03221=1152.962,292.404,-71.971,-177.029,8.258,148.750
C03222=1152.965,292.155,-71.940,-177.032,8.255,148.750
C03223=1152.970,291.907,-71.909,-177.035,8.252,148.750
C03224=1152.974,291.659,-71.880,-177.038,8.248,148.750
C03225=1152.979,291.411,-71.849,-177.040,8.245,148.750
C03226=1152.983,291.163,-71.820,-177.043,8.242,148.750
C03227=1152.987,290.915,-71.789,-177.045,8.239,148.750
C03228=1152.992,290.667,-71.759,-177.048,8.236,148.750
C03229=1152.996,290.419,-71.729,-177.050,8.233,148.750
C03230=1153.000,290.170,-71.699,-177.053,8.230,148.750
C03231=1153.004,289.922,-71.669,-177.055,8.227,148.749
C03232=1153.008,289.674,-71.639,-177.059,8.223,148.749
C03233=1153.013,289.426,-71.608,-177.062,8.220,148.749
C03234=1153.017,289.178,-71.579,-177.064,8.217,148.749
C03235=1153.021,288.930,-71.549,-177.067,8.214,148.749
C03236=1153.025,288.681,-71.519,-177.069,8.210,148.749
C03237=1153.029,288.434,-71.489,-177.072,8.207,148.749
C03238=1153.034,288.185,-71.459,-177.074,8.204,148.749
C03239=1153.038,287.910,-71.427,-177.077,8.200,148.749
C03240=1153.043,287.635,-71.393,-177.080,8.197,148.749
C03241=1153.048,287.359,-71.359,-177.083,8.194,148.749
C03242=1153.053,287.084,-71.326,-177.086,8.190,148.749
C03243=1153.057,286.836,-71.297,-177.089,8.187,148.749
C03244=1153.061,286.588,-71.267,-177.092,8.184,148.749
C03245=1153.065,286.340,-71.237,-177.094,8.180,148.749
C03246=1153.070,286.091,-71.207,-177.097,8.177,148.749
C03247=1153.074,285.844,-71.177,-177.099,8.174,148.749
C03248=1153.078,285.595,-71.148,-177.102,8.171,148.749
C03249=1153.082,285.347,-71.118,-177.105,8.168,148.749
C03250=1153.086,285.099,-71.089,-177.107,8.165,148.749
C03251=1153.091,284.850,-71.059,-177.111,8.161,148.749
C03252=1153.095,284.603,-71.028,-177.113,8.158,148.749
C03253=1153.099,284.354,-70.999,-177.116,8.155,148.748
C03254=1153.104,284.106,-70.970,-177.118,8.152,148.749
C03255=1153.108,283.858,-70.940,-177.121,8.149,148.749
C03256=1153.112,283.610,-70.911,-177.123,8.146,148.748
C03257=1153.117,283.361,-70.881,-177.126,8.143,148.748
C03258=1153.121,283.113,-70.851,-177.129,8.140,148.748
C03259=1153.125,282.865,-70.821,-177.131,8.137,148.748
C03260=1153.129,282.617,-70.792,-177.134,8.134,148.748
C03261=1153.133,282.369,-70.762,-177.136,8.130,148.748
C03262=1153.137,282.120,-70.733,-177.140,8.127,148.748
C03263=1153.142,281.872,-70.703,-177.142,8.124,148.748
C03264=1153.146,281.624,-70.674,-177.145,8.121,148.748
C03265=1153.150,281.375,-70.644,-177.148,8.118,148.748
C03266=1153.155,281.128,-70.615,-177.150,8.115,148.748
C03267=1153.160,280.879,-70.585,-177.153,8.112,148.748
C03268=1153.164,280.631,-70.556,-177.155,8.108,148.748
C03269=1153.168,280.383,-70.526,-177.158,8.105,148.748
C03270=1153.172,280.135,-70.497,-177.161,8.102,148.748
C03271=1153.176,279.886,-70.467,-177.163,8.099,148.748
C03272=1153.181,279.638,-70.438,-177.166,8.096,148.748
C03273=1153.185,279.389,-70.409,-177.169,8.093,148.748
C03274=1153.189,279.141,-70.380,-177.172,8.090,148.748
C03275=1153.194,278.893,-70.351,-177.174,8.087,148.748
C03276=1153.198,278.645,-70.322,-177.177,8.083,148.748
C03277=1153.202,278.397,-70.292,-177.180,8.080,148.748
C03278=1153.206,278.149,-70.263,-177.182,8.077,148.748
C03279=1153.210,277.901,-70.233,-177.185,8.074,148.748
C03280=1153.215,277.652,-70.205,-177.188,8.071,148.748
C03281=1153.219,277.403,-70.175,-177.191,8.068,148.748
C03282=1153.224,277.156,-70.146,-177.193,8.065,148.748
C03283=1153.228,276.908,-70.117,-177.196,8.062,148.748
C03284=1153.232,276.659,-70.088,-177.199,8.059,148.748
C03285=1153.236,276.410,-70.058,-177.201,8.056,148.748
C03286=1153.241,276.162,-70.029,-177.204,8.053,148.748
C03287=1153.245,275.915,-70.000,-177.206,8.050,148.748
C03288=1153.249,275.666,-69.972,-177.209,8.047,148.748
C03289=1153.253,275.418,-69.942,-177.212,8.044,148.748
C03290=1153.257,275.169,-69.913,-177.214,8.041,148.748
C03291=1153.262,274.921,-69.884,-177.217,8.038,148.748
C03292=1153.267,274.673,-69.855,-177.220,8.035,148.748
C03293=1153.270,274.425,-69.826,-177.223,8.032,148.748
C03294=1153.275,274.176,-69.797,-177.225,8.029,148.748
C03295=1153.279,273.928,-69.768,-177.228,8.026,148.748
C03296=1153.284,273.680,-69.740,-177.230,8.023,148.748
C03297=1153.288,273.431,-69.710,-177.233,8.020,148.748
C03298=1153.292,273.183,-69.681,-177.236,8.017,148.748
C03299=1153.296,272.935,-69.653,-177.239,8.013,148.748
C03300=1153.301,272.687,-69.623,-177.242,8.010,148.748
C03301=1153.305,272.438,-69.595,-177.244,8.007,148.748
C03302=1153.309,272.190,-69.566,-177.247,8.004,148.748
C03303=1153.313,271.941,-69.537,-177.249,8.001,148.748
C03304=1153.318,271.694,-69.508,-177.252,7.998,148.748
C03305=1153.322,271.445,-69.480,-177.255,7.995,148.748
C03306=1153.326,271.197,-69.450,-177.258,7.992,148.748
C03307=1153.331,270.949,-69.422,-177.261,7.989,148.748
C03308=1153.336,270.700,-69.393,-177.263,7.986,148.748
C03309=1153.339,270.452,-69.364,-177.266,7.983,148.748
C03310=1153.344,270.204,-69.336,-177.268,7.980,148.748
C03311=1153.348,269.955,-69.307,-177.271,7.977,148.748
C03312=1153.352,269.707,-69.278,-177.274,7.974,148.748
C03313=1153.357,269.459,-69.250,-177.277,7.971,148.748
C03314=1153.361,269.211,-69.221,-177.279,7.968,148.748
C03315=1153.365,268.962,-69.193,-177.282,7.965,148.748
C03316=1153.370,268.714,-69.164,-177.285,7.962,148.748
C03317=1153.374,268.466,-69.135,-177.287,7.959,148.748
C03318=1153.378,268.217,-69.107,-177.290,7.956,148.748
C03319=1153.383,267.969,-69.078,-177.293,7.953,148.748
C03320=1153.387,267.720,-69.050,-177.296,7.950,148.748
C03321=1153.392,267.472,-69.021,-177.298,7.947,148.748
C03322=1153.395,267.224,-68.993,-177.301,7.944,148.748
C03323=1153.400,266.975,-68.964,-177.304,7.941,148.748
C03324=1153.404,266.727,-68.936,-177.306,7.938,148.748
C03325=1153.408,266.479,-68.907,-177.309,7.935,148.748
C03326=1153.413,266.231,-68.879,-177.312,7.932,148.748
C03327=1153.417,265.982,-68.850,-177.315,7.929,148.748
C03328=1153.421,265.733,-68.822,-177.317,7.926,148.748
C03329=1153.426,265.485,-68.794,-177.320,7.923,148.748
C03330=1153.430,265.237,-68.766,-177.322,7.920,148.748
C03331=1153.435,264.988,-68.737,-177.325,7.917,148.748
C03332=1153.439,264.740,-68.709,-177.328,7.914,148.749
C03333=1153.443,264.492,-68.680,-177.331,7.911,148.749
C03334=1153.447,264.244,-68.652,-177.333,7.909,148.749
C03335=1153.452,263.996,-68.624,-177.336,7.906,148.749
C03336=1153.456,263.747,-68.595,-177.338,7.903,148.749
C03337=1153.461,263.498,-68.567,-177.341,7.900,148.749
C03338=1153.465,263.250,-68.539,-177.344,7.897,148.749
C03339=1153.469,263.001,-68.510,-177.346,7.894,148.749
C03340=1153.474,262.753,-68.482,-177.349,7.891,148.749
C03341=1153.477,262.505,-68.454,-177.352,7.888,148.749
C03342=1153.483,262.257,-68.426,-177.355,7.885,148.749
C03343=1153.487,261.983,-68.395,-177.358,7.881,148.749
C03344=1153.492,261.710,-68.365,-177.361,7.878,148.749
C03345=1153.497,261.436,-68.333,-177.364,7.875,148.749
C03346=1153.502,261.163,-68.303,-177.367,7.872,148.749
C03347=1153.506,260.914,-68.274,-177.370,7.869,148.749
C03348=1153.510,260.667,-68.247,-177.373,7.866,148.749
C03349=1153.515,260.418,-68.218,-177.375,7.864,148.749
C03350=1153.519,260.170,-68.190,-177.377,7.861,148.749
C03351=1153.523,259.921,-68.162,-177.380,7.858,148.749
C03352=1153.528,259.673,-68.134,-177.383,7.855,148.749
C03353=1153.532,259.425,-68.107,-177.386,7.852,148.750
C03354=1153.536,259.176,-68.078,-177.388,7.849,148.749
C03355=1153.540,258.928,-68.051,-177.391,7.846,148.749
C03356=1153.545,258.679,-68.022,-177.394,7.843,148.750
C03357=1153.550,258.431,-67.995,-177.396,7.840,148.750
C03358=1153.553,258.182,-67.967,-177.399,7.837,148.750
C03359=1153.558,257.934,-67.939,-177.402,7.834,148.750
C03360=1153.563,257.686,-67.911,-177.405,7.831,148.750
C03361=1153.567,257.437,-67.883,-177.408,7.828,148.750
C03362=1153.571,257.189,-67.855,-177.410,7.825,148.750
C03363=1153.575,256.940,-67.827,-177.413,7.822,148.750
C03364=1153.580,256.692,-67.800,-177.416,7.819,148.750
C03365=1153.585,256.444,-67.772,-177.418,7.817,148.750
C03366=1153.588,256.195,-67.744,-177.421,7.814,148.750
C03367=1153.593,255.947,-67.717,-177.424,7.811,148.750
C03368=1153.597,255.699,-67.689,-177.426,7.808,148.750
C03369=1153.602,255.450,-67.661,-177.429,7.805,148.750
C03370=1153.606,255.202,-67.634,-177.432,7.802,148.750
C03371=1153.611,254.954,-67.605,-177.435,7.800,148.751
C03372=1153.615,254.704,-67.578,-177.437,7.797,148.751
C03373=1153.619,254.457,-67.550,-177.440,7.794,148.751
C03374=1153.623,254.207,-67.523,-177.443,7.791,148.751
C03375=1153.628,253.959,-67.495,-177.446,7.788,148.751
C03376=1153.632,253.711,-67.468,-177.449,7.785,148.751
C03377=1153.637,253.463,-67.440,-177.451,7.783,148.751
C03378=1153.641,253.214,-67.413,-177.454,7.780,148.751
C03379=1153.645,252.966,-67.385,-177.456,7.777,148.751
C03380=1153.650,252.718,-67.358,-177.459,7.774,148.751
C03381=1153.654,252.469,-67.330,-177.462,7.771,148.751
C03382=1153.658,252.220,-67.302,-177.465,7.768,148.751
C03383=1153.663,251.972,-67.275,-177.467,7.765,148.751
C03384=1153.667,251.723,-67.247,-177.470,7.762,148.751
C03385=1153.672,251.475,-67.220,-177.473,7.759,148.751
C03386=1153.676,251.227,-67.192,-177.475,7.757,148.752
C03387=1153.681,250.978,-67.165,-177.478,7.754,148.752
C03388=1153.684,250.729,-67.138,-177.481,7.751,148.752
C03389=1153.689,250.481,-67.110,-177.484,7.748,148.752
C03390=1153.693,250.233,-67.083,-177.486,7.745,148.752
C03391=1153.698,249.984,-67.056,-177.489,7.742,148.752
C03392=1153.702,249.736,-67.028,-177.492,7.739,148.752
C03393=1153.706,249.487,-67.001,-177.495,7.737,148.752
C03394=1153.711,249.239,-66.974,-177.498,7.734,148.752
C03395=1153.716,248.990,-66.947,-177.500,7.732,148.752
C03396=1153.720,248.743,-66.919,-177.503,7.729,148.752
C03397=1153.724,248.493,-66.892,-177.506,7.726,148.753
C03398=1153.729,248.245,-66.864,-177.508,7.723,148.753
C03399=1153.733,247.996,-66.837,-177.511,7.720,148.753
C03400=1153.738,247.748,-66.810,-177.514,7.717,148.753
C03401=1153.743,247.500,-66.783,-177.517,7.714,148.753
C03402=1153.746,247.251,-66.756,-177.520,7.711,148.753
C03403=1153.750,247.003,-66.729,-177.522,7.709,148.753
C03404=1153.755,246.754,-66.702,-177.524,7.706,148.753
C03405=1153.760,246.506,-66.675,-177.527,7.703,148.753
C03406=1153.764,246.257,-66.647,-177.530,7.700,148.753
C03407=1153.769,246.009,-66.620,-177.533,7.698,148.754
C03408=1153.772,245.760,-66.594,-177.536,7.695,148.754
C03409=1153.777,245.511,-66.567,-177.539,7.692,148.754
C03410=1153.782,245.263,-66.539,-177.541,7.690,148.754
C03411=1153.786,245.015,-66.512,-177.544,7.687,148.754
C03412=1153.791,244.766,-66.485,-177.547,7.684,148.754
C03413=1153.795,244.518,-66.458,-177.549,7.681,148.754
C03414=1153.799,244.270,-66.431,-177.552,7.678,148.754
C03415=1153.803,244.020,-66.404,-177.555,7.675,148.754
C03416=1153.808,243.772,-66.377,-177.557,7.673,148.754
C03417=1153.812,243.523,-66.351,-177.560,7.670,148.755
C03418=1153.817,243.275,-66.324,-177.563,7.667,148.755
C03419=1153.822,243.026,-66.297,-177.566,7.664,148.755
C03420=1153.825,242.778,-66.270,-177.569,7.662,148.755
C03421=1153.830,242.529,-66.243,-177.571,7.659,148.755
C03422=1153.835,242.281,-66.216,-177.574,7.656,148.755
C03423=1153.839,242.033,-66.190,-177.576,7.654,148.755
C03424=1153.843,241.784,-66.163,-177.579,7.651,148.755
C03425=1153.848,241.536,-66.136,-177.582,7.648,148.755
C03426=1153.852,241.288,-66.109,-177.585,7.645,148.755
C03427=1153.857,241.039,-66.083,-177.588,7.642,148.756
C03428=1153.861,240.789,-66.055,-177.590,7.640,148.756
C03429=1153.865,240.541,-66.029,-177.593,7.637,148.756
C03430=1153.870,240.293,-66.002,-177.596,7.634,148.756
C03431=1153.874,240.044,-65.975,-177.599,7.631,148.756
C03432=1153.878,239.795,-65.949,-177.602,7.629,148.756
C03433=1153.883,239.547,-65.922,-177.604,7.627,148.756
C03434=1153.887,239.299,-65.895,-177.607,7.624,148.756
C03435=1153.892,239.050,-65.868,-177.610,7.621,148.756
C03436=1153.897,238.801,-65.842,-177.612,7.618,148.756
C03437=1153.901,238.553,-65.816,-177.615,7.615,148.757
C03438=1153.905,238.304,-65.789,-177.617,7.613,148.757
C03439=1153.909,238.056,-65.763,-177.621,7.610,148.757
C03440=1153.914,237.807,-65.736,-177.623,7.607,148.757
C03441=1153.918,237.559,-65.709,-177.626,7.604,148.757
C03442=1153.923,237.310,-65.683,-177.629,7.601,148.757
C03443=1153.927,237.062,-65.656,-177.631,7.599,148.757
C03444=1153.932,236.813,-65.630,-177.634,7.597,148.758
C03445=1153.936,236.565,-65.604,-177.637,7.594,148.758
C03446=1153.941,236.316,-65.577,-177.640,7.591,148.758
C03447=1153.945,236.044,-65.549,-177.643,7.588,148.758
C03448=1153.950,235.772,-65.519,-177.646,7.585,148.758
C03449=1153.956,235.500,-65.491,-177.649,7.582,148.758
C03450=1153.960,235.229,-65.462,-177.652,7.579,148.758
C03451=1153.964,234.981,-65.435,-177.654,7.576,148.758
C03452=1153.969,234.731,-65.409,-177.658,7.574,148.759
C03453=1153.973,234.483,-65.382,-177.660,7.571,148.759
C03454=1153.978,234.235,-65.357,-177.663,7.568,148.759
C03455=1153.983,233.986,-65.331,-177.665,7.566,148.759
C03456=1153.987,233.738,-65.304,-177.668,7.563,148.759
C03457=1153.992,233.489,-65.278,-177.671,7.560,148.759
C03458=1153.995,233.241,-65.251,-177.674,7.557,148.759
C03459=1154.000,232.991,-65.225,-177.676,7.555,148.759
C03460=1154.004,232.743,-65.199,-177.679,7.552,148.760
C03461=1154.009,232.494,-65.173,-177.682,7.549,148.760
C03462=1154.014,232.245,-65.147,-177.685,7.547,148.760
C03463=1154.018,231.998,-65.120,-177.687,7.545,148.760
C03464=1154.022,231.749,-65.095,-177.690,7.542,148.760
C03465=1154.027,231.500,-65.068,-177.693,7.539,148.760
C03466=1154.031,231.252,-65.042,-177.696,7.536,148.761
C03467=1154.035,231.003,-65.016,-177.698,7.534,148.761
C03468=1154.040,230.754,-64.990,-177.701,7.531,148.761
C03469=1154.045,230.506,-64.964,-177.704,7.528,148.761
C03470=1154.049,230.258,-64.938,-177.707,7.526,148.761
C03471=1154.053,230.009,-64.912,-177.709,7.524,148.761
C03472=1154.058,229.760,-64.886,-177.712,7.521,148.761
C03473=1154.062,229.511,-64.860,-177.715,7.518,148.761
C03474=1154.067,229.263,-64.834,-177.718,7.515,148.762
C03475=1154.071,229.015,-64.808,-177.720,7.513,148.762
C03476=1154.076,228.765,-64.782,-177.723,7.510,148.762
C03477=1154.080,228.517,-64.756,-177.726,7.507,148.762
C03478=1154.085,228.268,-64.730,-177.729,7.505,148.762
C03479=1154.089,228.020,-64.704,-177.731,7.502,148.762
C03480=1154.094,227.771,-64.678,-177.734,7.499,148.762
C03481=1154.098,227.522,-64.652,-177.737,7.497,148.763
C03482=1154.103,227.274,-64.626,-177.740,7.495,148.763
C03483=1154.107,227.026,-64.601,-177.742,7.492,148.763
C03484=1154.112,226.777,-64.575,-177.745,7.489,148.763
C03485=1154.116,226.528,-64.550,-177.748,7.486,148.763
C03486=1154.120,226.279,-64.524,-177.751,7.484,148.763
C03487=1154.126,226.031,-64.498,-177.753,7.481,148.764
C03488=1154.130,225.782,-64.472,-177.756,7.478,148.764
C03489=1154.134,225.533,-64.446,-177.759,7.477,148.764
C03490=1154.138,225.284,-64.421,-177.762,7.474,148.764
C03491=1154.143,225.036,-64.395,-177.764,7.471,148.764
C03492=1154.147,224.787,-64.369,-177.767,7.469,148.764
C03493=1154.152,224.539,-64.344,-177.770,7.466,148.765
C03494=1154.156,224.290,-64.318,-177.773,7.463,148.765
C03495=1154.161,224.042,-64.293,-177.775,7.460,148.765
C03496=1154.165,223.793,-64.267,-177.778,7.458,148.765
C03497=1154.170,223.545,-64.241,-177.781,7.455,148.765
C03498=1154.175,223.296,-64.215,-177.784,7.453,148.765
C03499=1154.179,223.047,-64.189,-177.786,7.451,148.766
C03500=1154.184,222.799,-64.164,-177.789,7.448,148.766
C03501=1154.188,222.550,-64.138,-177.792,7.445,148.766
C03502=1154.192,222.300,-64.113,-177.795,7.443,148.766
C03503=1154.197,222.052,-64.088,-177.797,7.440,148.766
C03504=1154.202,221.804,-64.062,-177.800,7.437,148.766
C03505=1154.206,221.555,-64.036,-177.803,7.436,148.767
C03506=1154.211,221.307,-64.011,-177.806,7.433,148.767
C03507=1154.215,221.057,-63.986,-177.808,7.430,148.767
C03508=1154.219,220.809,-63.961,-177.811,7.428,148.767
C03509=1154.223,220.561,-63.935,-177.814,7.425,148.767
C03510=1154.228,220.312,-63.910,-177.817,7.422,148.767
C03511=1154.233,220.063,-63.885,-177.819,7.420,148.768
C03512=1154.237,219.814,-63.859,-177.822,7.417,148.768
C03513=1154.242,219.566,-63.834,-177.825,7.414,148.768
C03514=1154.246,219.317,-63.808,-177.828,7.413,148.768
C03515=1154.251,219.068,-63.783,-177.830,7.410,148.768
C03516=1154.255,218.820,-63.758,-177.833,7.407,148.768
C03517=1154.260,218.571,-63.732,-177.836,7.405,148.769
C03518=1154.264,218.323,-63.708,-177.839,7.402,148.769
C03519=1154.268,218.074,-63.682,-177.841,7.399,148.769
C03520=1154.272,217.825,-63.656,-177.844,7.397,148.769
C03521=1154.278,217.576,-63.632,-177.847,7.394,148.769
C03522=1154.282,217.328,-63.606,-177.850,7.392,148.769
C03523=1154.287,217.079,-63.581,-177.852,7.390,148.770
C03524=1154.291,216.830,-63.555,-177.855,7.387,148.770
C03525=1154.296,216.582,-63.531,-177.858,7.384,148.770
C03526=1154.300,216.333,-63.506,-177.861,7.382,148.770
C03527=1154.305,216.085,-63.480,-177.863,7.379,148.770
C03528=1154.309,215.835,-63.455,-177.866,7.377,148.771
C03529=1154.313,215.587,-63.430,-177.869,7.375,148.771
C03530=1154.318,215.338,-63.405,-177.872,7.372,148.771
C03531=1154.323,215.090,-63.380,-177.874,7.370,148.771
C03532=1154.327,214.841,-63.355,-177.877,7.367,148.771
C03533=1154.332,214.592,-63.331,-177.880,7.364,148.772
C03534=1154.336,214.343,-63.305,-177.883,7.362,148.772
C03535=1154.341,214.095,-63.280,-177.885,7.359,148.772
C03536=1154.345,213.846,-63.255,-177.888,7.358,148.772
C03537=1154.349,213.597,-63.231,-177.891,7.355,148.772
C03538=1154.354,213.349,-63.205,-177.894,7.352,148.773
C03539=1154.359,213.100,-63.180,-177.896,7.350,148.773
C03540=1154.363,212.851,-63.156,-177.899,7.347,148.773
C03541=1154.367,212.603,-63.130,-177.902,7.345,148.773
C03542=1154.372,212.353,-63.105,-177.904,7.342,148.773
C03543=1154.376,212.105,-63.081,-177.908,7.340,148.774
C03544=1154.381,211.857,-63.056,-177.910,7.338,148.774
C03545=1154.386,211.607,-63.031,-177.913,7.335,148.774
C03546=1154.390,211.359,-63.007,-177.915,7.333,148.774
C03547=1154.395,211.109,-62.982,-177.918,7.330,148.774
C03548=1154.399,210.861,-62.956,-177.921,7.327,148.775
C03549=1154.404,210.613,-62.932,-177.924,7.325,148.775
C03550=1154.408,210.363,-62.907,-177.927,7.323,148.775
C03551=1154.414,210.093,-62.881,-177.930,7.320,148.775
C03552=1154.418,209.822,-62.853,-177.933,7.317,148.775
C03553=1154.423,209.552,-62.827,-177.935,7.315,148.776
C03554=1154.428,209.281,-62.800,-177.938,7.313,148.776
C03555=1154.433,209.033,-62.775,-177.941,7.310,148.776
C03556=1154.437,208.784,-62.751,-177.944,7.308,148.776
C03557=1154.442,208.535,-62.725,-177.947,7.305,148.776
C03558=1154.446,208.287,-62.701,-177.950,7.302,148.777
C03559=1154.451,208.038,-62.676,-177.952,7.300,148.777
C03560=1154.455,207.789,-62.652,-177.955,7.298,148.777
C03561=1154.460,207.540,-62.627,-177.958,7.296,148.777
C03562=1154.464,207.291,-62.603,-177.960,7.293,148.777
C03563=1154.469,207.043,-62.578,-177.963,7.291,148.778
C03564=1154.473,206.794,-62.554,-177.966,7.288,148.778
C03565=1154.478,206.545,-62.529,-177.969,7.285,148.778
C03566=1154.482,206.296,-62.505,-177.971,7.283,148.778
C03567=1154.487,206.048,-62.480,-177.975,7.281,148.779
C03568=1154.492,205.799,-62.456,-177.977,7.279,148.779
C03569=1154.496,205.550,-62.431,-177.980,7.276,148.779
C03570=1154.501,205.301,-62.407,-177.982,7.274,148.779
C03571=1154.506,205.053,-62.382,-177.986,7.271,148.779
C03572=1154.510,204.804,-62.358,-177.988,7.269,148.780
C03573=1154.514,204.555,-62.334,-177.991,7.267,148.780
C03574=1154.519,204.306,-62.309,-177.993,7.265,148.780
C03575=1154.524,204.058,-62.285,-177.996,7.262,148.780
C03576=1154.528,203.809,-62.260,-177.999,7.259,148.780
C03577=1154.532,203.560,-62.236,-178.002,7.257,148.781
C03578=1154.537,203.312,-62.212,-178.005,7.254,148.781
C03579=1154.542,203.063,-62.187,-178.007,7.253,148.781
C03580=1154.546,202.814,-62.163,-178.010,7.250,148.781
C03581=1154.551,202.565,-62.140,-178.013,7.248,148.782
C03582=1154.556,202.316,-62.115,-178.016,7.245,148.782
C03583=1154.560,202.068,-62.091,-178.018,7.243,148.782
C03584=1154.564,201.819,-62.066,-178.021,7.240,148.782
C03585=1154.569,201.570,-62.042,-178.024,7.239,148.783
C03586=1154.574,201.321,-62.018,-178.027,7.236,148.783
C03587=1154.578,201.072,-61.994,-178.029,7.234,148.783
C03588=1154.583,200.824,-61.970,-178.032,7.231,148.783
C03589=1154.587,200.575,-61.945,-178.035,7.229,148.784
C03590=1154.592,200.326,-61.922,-178.038,7.226,148.784
C03591=1154.596,200.077,-61.898,-178.040,7.225,148.784
C03592=1154.601,199.828,-61.873,-178.043,7.222,148.784
C03593=1154.606,199.580,-61.849,-178.046,7.220,148.784
C03594=1154.610,199.330,-61.825,-178.049,7.217,148.785
C03595=1154.614,199.082,-61.801,-178.051,7.215,148.785
C03596=1154.619,198.833,-61.777,-178.054,7.212,148.785
C03597=1154.624,198.584,-61.753,-178.057,7.211,148.785
C03598=1154.628,198.336,-61.729,-178.060,7.208,148.786
C03599=1154.633,198.087,-61.705,-178.062,7.206,148.786
C03600=1154.637,197.838,-61.681,-178.065,7.203,148.786
C03601=1154.642,197.589,-61.657,-178.068,7.201,148.786
C03602=1154.647,197.340,-61.633,-178.071,7.199,148.787
C03603=1154.651,197.091,-61.609,-178.073,7.197,148.787
C03604=1154.655,196.843,-61.585,-178.076,7.194,148.787
C03605=1154.660,196.594,-61.562,-178.079,7.192,148.787
C03606=1154.665,196.346,-61.538,-178.082,7.189,148.788
C03607=1154.669,196.097,-61.514,-178.084,7.187,148.788
C03608=1154.674,195.848,-61.490,-178.087,7.185,148.788
C03609=1154.678,195.598,-61.466,-178.090,7.183,148.788
C03610=1154.683,195.350,-61.442,-178.093,7.180,148.788
C03611=1154.688,195.101,-61.419,-178.095,7.178,148.789
C03612=1154.692,194.852,-61.394,-178.098,7.175,148.789
C03613=1154.697,194.603,-61.371,-178.101,7.174,148.789
C03614=1154.701,194.355,-61.347,-178.103,7.171,148.789
C03615=1154.706,194.106,-61.324,-178.106,7.169,148.790
C03616=1154.710,193.857,-61.300,-178.109,7.167,148.790
C03617=1154.715,193.608,-61.276,-178.112,7.164,148.790
C03618=1154.720,193.359,-61.253,-178.115,7.162,148.791
C03619=1154.724,193.111,-61.229,-178.117,7.159,148.791
C03620=1154.729,192.862,-61.205,-178.120,7.158,148.791
C03621=1154.733,192.613,-61.182,-178.123,7.155,148.791
C03622=1154.738,192.364,-61.158,-178.126,7.153,148.792
C03623=1154.742,192.115,-61.135,-178.129,7.150,148.792
C03624=1154.747,191.866,-61.111,-178.131,7.148,148.792
C03625=1154.752,191.618,-61.087,-178.134,7.147,148.792
C03626=1154.756,191.369,-61.064,-178.137,7.144,148.793
C03627=1154.761,191.120,-61.040,-178.139,7.142,148.793
C03628=1154.766,190.871,-61.017,-178.142,7.139,148.793
C03629=1154.770,190.622,-60.993,-178.145,7.137,148.793
C03630=1154.775,190.373,-60.970,-178.148,7.135,148.794
C03631=1154.779,190.124,-60.946,-178.151,7.133,148.794
C03632=1154.784,189.875,-60.923,-178.153,7.130,148.794
C03633=1154.788,189.627,-60.899,-178.156,7.128,148.794
C03634=1154.793,189.378,-60.876,-178.159,7.127,148.795
C03635=1154.798,189.129,-60.852,-178.162,7.124,148.795
C03636=1154.803,188.880,-60.829,-178.164,7.122,148.795
C03637=1154.807,188.631,-60.805,-178.167,7.119,148.795
C03638=1154.812,188.382,-60.782,-178.170,7.117,148.796
C03639=1154.816,188.134,-60.759,-178.172,7.115,148.796
C03640=1154.820,187.885,-60.735,-178.175,7.113,148.796
C03641=1154.825,187.636,-60.712,-178.178,7.111,148.797
C03642=1154.830,187.387,-60.689,-178.181,7.108,148.797
C03643=1154.834,187.137,-60.665,-178.183,7.106,148.797
C03644=1154.840,186.889,-60.642,-178.187,7.104,148.797
C03645=1154.844,186.640,-60.619,-178.189,7.101,148.797
C03646=1154.848,186.391,-60.596,-178.192,7.100,148.798
C03647=1154.853,186.142,-60.573,-178.195,7.097,148.798
C03648=1154.858,185.893,-60.549,-178.197,7.095,148.798
C03649=1154.863,185.644,-60.526,-178.200,7.093,148.799
C03650=1154.867,185.395,-60.503,-178.203,7.091,148.799
C03651=1154.871,185.147,-60.480,-178.205,7.089,148.799
C03652=1154.876,184.898,-60.457,-178.209,7.086,148.800
C03653=1154.881,184.648,-60.433,-178.211,7.084,148.800
